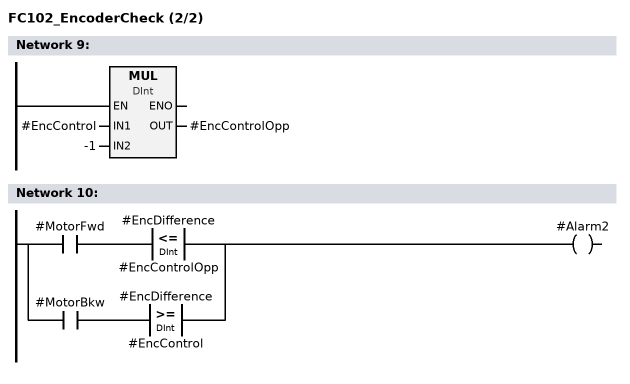
   RUNG wire#powerrail
      { S7_Templates := "SrcType := DInt"; S7_GenerateENO := "TRUE" } Mul(in1 := #EncControl, in2 := -1, out => #EncControlOpp)
   END_RUNG
   // the same network as SCL:
   #EncControlOpp := #EncControl * (-1);
END_REGION

REGION Network 10
   RUNG wire#powerrail
      Contact( #MotorFwd )
      { S7_Templates := "SrcType := DInt" } LE_Contact(in1 := #EncDifference, in2 := #EncControlOpp)
      wire#w1
      Coil( #Alarm2 )
   END_RUNG
   RUNG wire#powerrail
      Contact( #MotorBkw )
      { S7_Templates := "SrcType := DInt" } GE_Contact(in1 := #EncDifference, in2 := #EncControl)
   END_RUNG wire#w1
   // the same network as SCL:
   #Alarm2 := (#MotorFwd AND (#EncDifference <= #EncControlOpp)) OR (#MotorBkw AND (#EncDifference >= #EncControl));
END_REGION
END_FUNCTION

FUNCTION "FC06_TechnoplatCycle" : Void   // FC6, LAD
TITLE = Machine cycle
{ S7_Optimized_Access := 'FALSE' }
AUTHOR : Robopac
VERSION : 0.0
// stored: AutoNumber false, IsIECCheckEnabled false, SetENOAutomatically false, UDAEnableTagReadback false
   VAR_TEMP   // added for the SCL form of the ladder/FBD networks
      _w1 : Bool;
   END_VAR
BEGIN

REGION Network 1: Machine cycle: M0.0 Start cycle
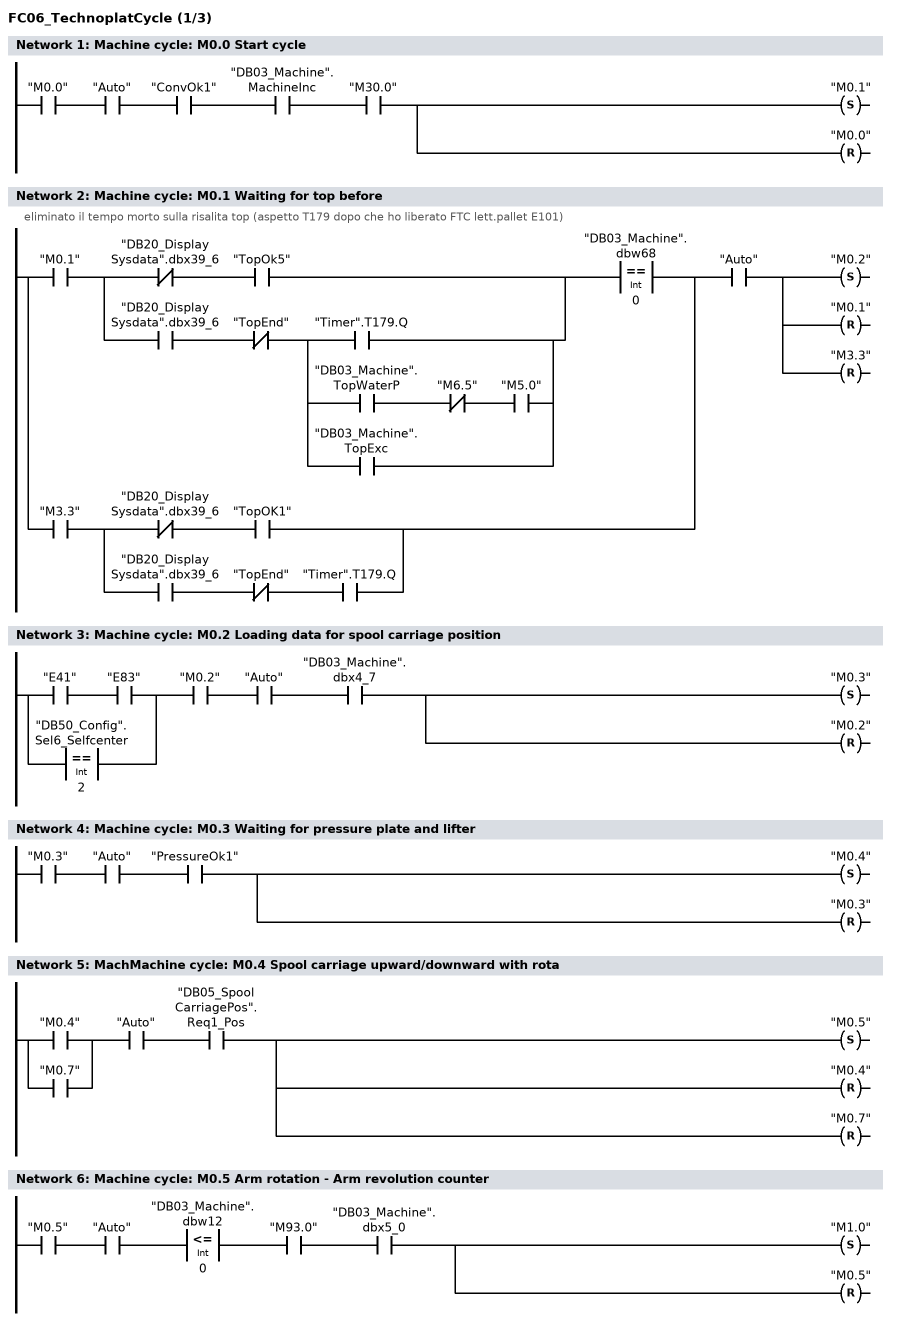
   RUNG wire#powerrail
      Contact( "M0.0" )
      Contact( "Auto" )
      Contact( "ConvOk1" )
      Contact( "DB03_Machine".MachineInc )
      Contact( "M30.0" )
      wire#w1
      S_Coil( "M0.1" )
   END_RUNG
   RUNG wire#w1
      R_Coil( "M0.0" )
   END_RUNG
   // the same network as SCL:
   IF "M0.0" AND "Auto" AND "ConvOk1" AND "DB03_Machine".MachineInc AND "M30.0" THEN
       "M0.1" := TRUE;
       "M0.0" := FALSE;
   END_IF;
END_REGION

REGION Network 2: Machine cycle: M0.1 Waiting for top before
   // eliminato il tempo morto sulla risalita top (aspetto T179 dopo che ho liberato FTC lett.pallet E101)
   RUNG wire#powerrail
      Contact( "M0.1" )
      wire#w1
      I_Contact( "DB20_DisplaySysdata".dbx39_6 )
      Contact( "TopOk5" )
      wire#w2
      { S7_Templates := "SrcType := Int" } EQ_Contact(in1 := "DB03_Machine".dbw68, in2 := 0)
      wire#w4
      Contact( "Auto" )
      wire#w6
      S_Coil( "M0.2" )
   END_RUNG
   RUNG wire#w1
      Contact( "DB20_DisplaySysdata".dbx39_6 )
      I_Contact( "TopEnd" )
      wire#w3
      Contact( "Timer".T179.Q )
   END_RUNG wire#w2
   RUNG wire#w3
      Contact( "DB03_Machine".TopWaterP )
      I_Contact( "M6.5" )
      Contact( "M5.0" )
   END_RUNG wire#w2
   RUNG wire#w3
      Contact( "DB03_Machine".TopExc )
   END_RUNG wire#w2
   RUNG wire#powerrail
      Contact( "M3.3" )
      wire#w5
      I_Contact( "DB20_DisplaySysdata".dbx39_6 )
      Contact( "TopOK1" )
   END_RUNG wire#w4
   RUNG wire#w5
      Contact( "DB20_DisplaySysdata".dbx39_6 )
      I_Contact( "TopEnd" )
      Contact( "Timer".T179.Q )
   END_RUNG wire#w4
   RUNG wire#w6
      R_Coil( "M0.1" )
   END_RUNG
   RUNG wire#w6
      R_Coil( "M3.3" )
   END_RUNG
   // the same network as SCL:
   IF (("M0.1" AND ((NOT "DB20_DisplaySysdata".dbx39_6 AND "TopOk5") OR ("DB20_DisplaySysdata".dbx39_6 AND NOT "TopEnd" AND ("Timer".T179.Q OR ("DB03_Machine".TopWaterP AND NOT "M6.5" AND "M5.0") OR "DB03_Machine".TopExc))) AND ("DB03_Machine".dbw68 = 0)) OR ("M3.3" AND ((NOT "DB20_DisplaySysdata".dbx39_6 AND "TopOK1") OR ("DB20_DisplaySysdata".dbx39_6 AND NOT "TopEnd" AND "Timer".T179.Q)))) AND "Auto" THEN
       "M0.2" := TRUE;
   END_IF;
   #_w1 := (("M0.1" AND ((NOT "DB20_DisplaySysdata".dbx39_6 AND "TopOk5") OR ("DB20_DisplaySysdata".dbx39_6 AND NOT "TopEnd" AND ("Timer".T179.Q OR ("DB03_Machine".TopWaterP AND NOT "M6.5" AND "M5.0") OR "DB03_Machine".TopExc))) AND ("DB03_Machine".dbw68 = 0)) OR ("M3.3" AND ((NOT "DB20_DisplaySysdata".dbx39_6 AND "TopOK1") OR ("DB20_DisplaySysdata".dbx39_6 AND NOT "TopEnd" AND "Timer".T179.Q)))) AND "Auto";
   IF #_w1 THEN
       "M0.1" := FALSE;
       "M3.3" := FALSE;
   END_IF;
END_REGION

REGION Network 3: Machine cycle: M0.2 Loading data for spool carriage position
   RUNG wire#powerrail
      Contact( "E41" )
      Contact( "E83" )
      wire#w1
      Contact( "M0.2" )
      Contact( "Auto" )
      Contact( "DB03_Machine".dbx4_7 )
      wire#w2
      S_Coil( "M0.3" )
   END_RUNG
   RUNG wire#powerrail
      { S7_Templates := "SrcType := Int" } EQ_Contact(in1 := "DB50_Config".Sel6_Selfcenter, in2 := 2)
   END_RUNG wire#w1
   RUNG wire#w2
      R_Coil( "M0.2" )
   END_RUNG
   // the same network as SCL:
   IF (("E41" AND "E83") OR ("DB50_Config".Sel6_Selfcenter = 2)) AND "M0.2" AND "Auto" AND "DB03_Machine".dbx4_7 THEN
       "M0.3" := TRUE;
       "M0.2" := FALSE;
   END_IF;
END_REGION

REGION Network 4: Machine cycle: M0.3 Waiting for pressure plate and lifter
   RUNG wire#powerrail
      Contact( "M0.3" )
      Contact( "Auto" )
      Contact( "PressureOk1" )
      wire#w1
      S_Coil( "M0.4" )
   END_RUNG
   RUNG wire#w1
      R_Coil( "M0.3" )
   END_RUNG
   // the same network as SCL:
   IF "M0.3" AND "Auto" AND "PressureOk1" THEN
       "M0.4" := TRUE;
       "M0.3" := FALSE;
   END_IF;
END_REGION

REGION Network 5: MachMachine cycle: M0.4 Spool carriage upward/downward with rota
   RUNG wire#powerrail
      Contact( "M0.4" )
      wire#w1
      Contact( "Auto" )
      Contact( "DB05_SpoolCarriagePos".Req1_Pos )
      wire#w2
      S_Coil( "M0.5" )
   END_RUNG
   RUNG wire#powerrail
      Contact( "M0.7" )
   END_RUNG wire#w1
   RUNG wire#w2
      R_Coil( "M0.4" )
   END_RUNG
   RUNG wire#w2
      R_Coil( "M0.7" )
   END_RUNG
   // the same network as SCL:
   IF ("M0.4" OR "M0.7") AND "Auto" AND "DB05_SpoolCarriagePos".Req1_Pos THEN "M0.5" := TRUE; END_IF;
   #_w1 := ("M0.4" OR "M0.7") AND "Auto" AND "DB05_SpoolCarriagePos".Req1_Pos;
   IF #_w1 THEN
       "M0.4" := FALSE;
       "M0.7" := FALSE;
   END_IF;
END_REGION

REGION Network 6: Machine cycle: M0.5 Arm rotation - Arm revolution counter
   RUNG wire#powerrail
      Contact( "M0.5" )
      Contact( "Auto" )
      { S7_Templates := "SrcType := Int" } LE_Contact(in1 := "DB03_Machine".dbw12, in2 := 0)
      Contact( "M93.0" )
      Contact( "DB03_Machine".dbx5_0 )
      wire#w1
      S_Coil( "M1.0" )
   END_RUNG
   RUNG wire#w1
      R_Coil( "M0.5" )
   END_RUNG
   // the same network as SCL:
   IF "M0.5" AND "Auto" AND ("DB03_Machine".dbw12 <= 0) AND "M93.0" AND "DB03_Machine".dbx5_0 THEN
       "M1.0" := TRUE;
       "M0.5" := FALSE;
   END_IF;
END_REGION

REGION Network 7: Machine cycle: M1.0 Revolution over welder contrast
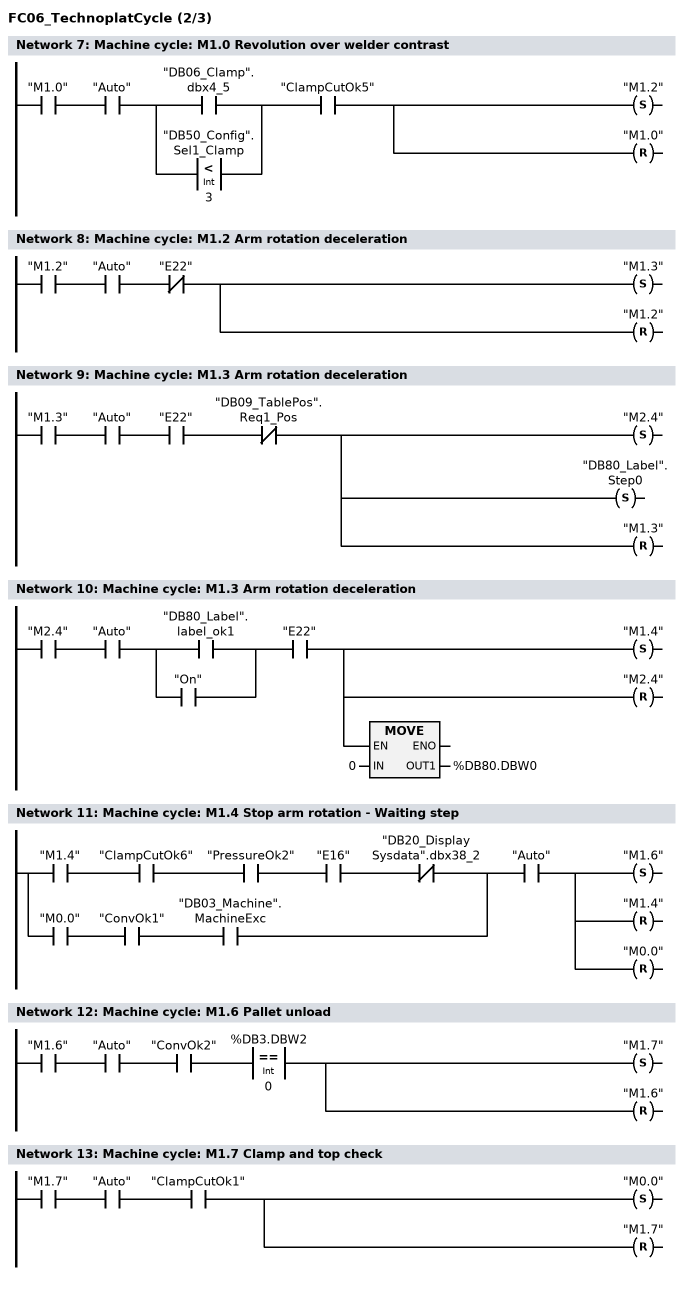
   RUNG wire#powerrail
      Contact( "M1.0" )
      Contact( "Auto" )
      wire#w1
      Contact( "DB06_Clamp".dbx4_5 )
      wire#w2
      Contact( "ClampCutOk5" )
      wire#w3
      S_Coil( "M1.2" )
   END_RUNG
   RUNG wire#w1
      { S7_Templates := "SrcType := Int" } LT_Contact(in1 := "DB50_Config".Sel1_Clamp, in2 := 3)
   END_RUNG wire#w2
   RUNG wire#w3
      R_Coil( "M1.0" )
   END_RUNG
   // the same network as SCL:
   IF "M1.0" AND "Auto" AND ("DB06_Clamp".dbx4_5 OR ("DB50_Config".Sel1_Clamp < 3)) AND "ClampCutOk5" THEN
       "M1.2" := TRUE;
       "M1.0" := FALSE;
   END_IF;
END_REGION

REGION Network 8: Machine cycle: M1.2 Arm rotation deceleration
   RUNG wire#powerrail
      Contact( "M1.2" )
      Contact( "Auto" )
      I_Contact( "E22" )
      wire#w1
      S_Coil( "M1.3" )
   END_RUNG
   RUNG wire#w1
      R_Coil( "M1.2" )
   END_RUNG
   // the same network as SCL:
   IF "M1.2" AND "Auto" AND NOT "E22" THEN
       "M1.3" := TRUE;
       "M1.2" := FALSE;
   END_IF;
END_REGION

REGION Network 9: Machine cycle: M1.3 Arm rotation deceleration
   RUNG wire#powerrail
      Contact( "M1.3" )
      Contact( "Auto" )
      Contact( "E22" )
      I_Contact( "DB09_TablePos".Req1_Pos )
      wire#w1
      S_Coil( "M2.4" )
   END_RUNG
   RUNG wire#w1
      S_Coil( "DB80_Label".Step0 )
   END_RUNG
   RUNG wire#w1
      R_Coil( "M1.3" )
   END_RUNG
   // the same network as SCL:
   IF "M1.3" AND "Auto" AND "E22" AND NOT "DB09_TablePos".Req1_Pos THEN
       "M2.4" := TRUE;
       "DB80_Label".Step0 := TRUE;
       "M1.3" := FALSE;
   END_IF;
END_REGION

REGION Network 10: Machine cycle: M1.3 Arm rotation deceleration
   RUNG wire#powerrail
      Contact( "M2.4" )
      Contact( "Auto" )
      wire#w1
      Contact( "DB80_Label".label_ok1 )
      wire#w2
      Contact( "E22" )
      wire#w3
      S_Coil( "M1.4" )
   END_RUNG
   RUNG wire#w1
      Contact( "On" )
   END_RUNG wire#w2
   RUNG wire#w3
      R_Coil( "M2.4" )
   END_RUNG
   RUNG wire#w3
      { S7_GenerateENO := "TRUE" } Move(in := 0, out1 => %DB80.DBW0)
   END_RUNG
   // the same network as SCL:
   IF "M2.4" AND "Auto" AND ("DB80_Label".label_ok1 OR "On") AND "E22" THEN "M1.4" := TRUE; END_IF;
   #_w1 := "M2.4" AND "Auto" AND ("DB80_Label".label_ok1 OR "On") AND "E22";
   IF #_w1 THEN
       "M2.4" := FALSE;
       %DB80.DBW0 := 0;
   END_IF;
END_REGION

REGION Network 11: Machine cycle: M1.4 Stop arm rotation - Waiting step
   RUNG wire#powerrail
      Contact( "M1.4" )
      Contact( "ClampCutOk6" )
      Contact( "PressureOk2" )
      Contact( "E16" )
      I_Contact( "DB20_DisplaySysdata".dbx38_2 )
      wire#w1
      Contact( "Auto" )
      wire#w2
      S_Coil( "M1.6" )
   END_RUNG
   RUNG wire#powerrail
      Contact( "M0.0" )
      Contact( "ConvOk1" )
      Contact( "DB03_Machine".MachineExc )
   END_RUNG wire#w1
   RUNG wire#w2
      R_Coil( "M1.4" )
   END_RUNG
   RUNG wire#w2
      R_Coil( "M0.0" )
   END_RUNG
   // the same network as SCL:
   IF (("M1.4" AND "ClampCutOk6" AND "PressureOk2" AND "E16" AND NOT "DB20_DisplaySysdata".dbx38_2) OR ("M0.0" AND "ConvOk1" AND "DB03_Machine".MachineExc)) AND "Auto" THEN
       "M1.6" := TRUE;
   END_IF;
   #_w1 := (("M1.4" AND "ClampCutOk6" AND "PressureOk2" AND "E16" AND NOT "DB20_DisplaySysdata".dbx38_2) OR ("M0.0" AND "ConvOk1" AND "DB03_Machine".MachineExc)) AND "Auto";
   IF #_w1 THEN
       "M1.4" := FALSE;
       "M0.0" := FALSE;
   END_IF;
END_REGION

REGION Network 12: Machine cycle: M1.6 Pallet unload
   RUNG wire#powerrail
      Contact( "M1.6" )
      Contact( "Auto" )
      Contact( "ConvOk2" )
      { S7_Templates := "SrcType := Int" } EQ_Contact(in1 := %DB3.DBW2, in2 := 0)
      wire#w1
      S_Coil( "M1.7" )
   END_RUNG
   RUNG wire#w1
      R_Coil( "M1.6" )
   END_RUNG
   // the same network as SCL:
   IF "M1.6" AND "Auto" AND "ConvOk2" AND (%DB3.DBW2 = 0) THEN
       "M1.7" := TRUE;
       "M1.6" := FALSE;
   END_IF;
END_REGION

REGION Network 13: Machine cycle: M1.7 Clamp and top check
   RUNG wire#powerrail
      Contact( "M1.7" )
      Contact( "Auto" )
      Contact( "ClampCutOk1" )
      wire#w1
      S_Coil( "M0.0" )
   END_RUNG
   RUNG wire#w1
      R_Coil( "M1.7" )
   END_RUNG
   // the same network as SCL:
   IF "M1.7" AND "Auto" AND "ClampCutOk1" THEN
       "M0.0" := TRUE;
       "M1.7" := FALSE;
   END_IF;
END_REGION

REGION Network 14: Machine cycle: M0.5 Arm rotation - Arm revolution counter
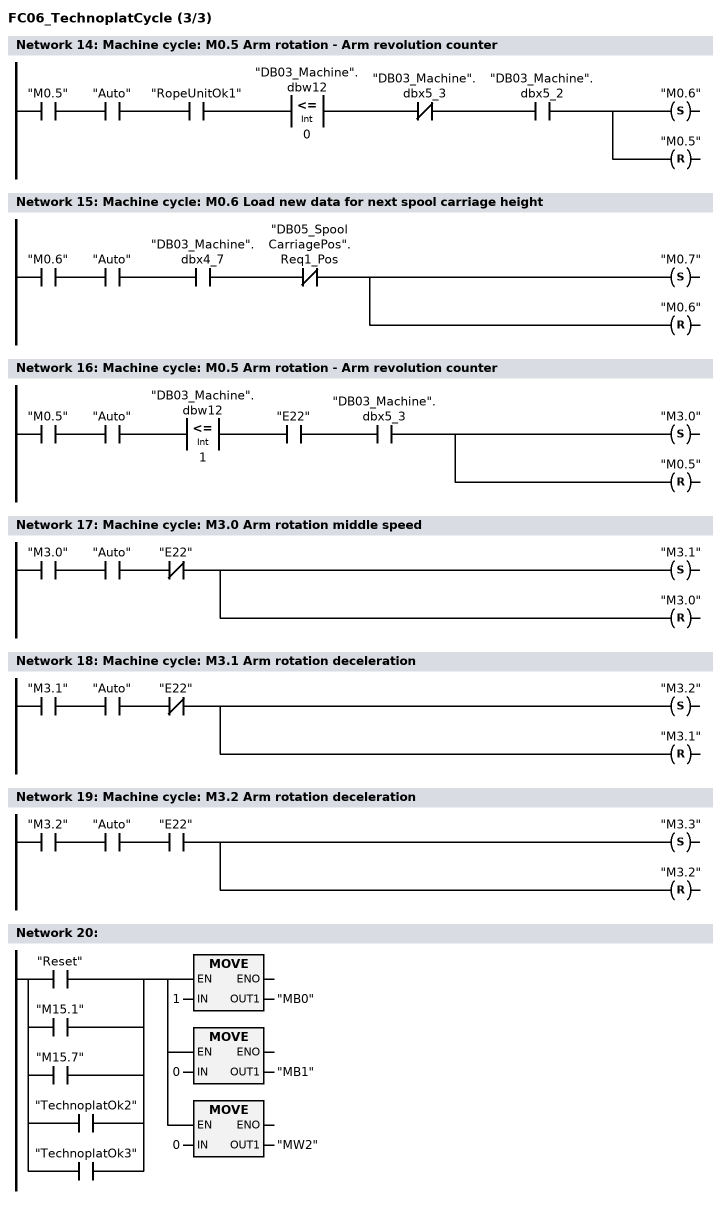
   RUNG wire#powerrail
      Contact( "M0.5" )
      Contact( "Auto" )
      Contact( "RopeUnitOk1" )
      { S7_Templates := "SrcType := Int" } LE_Contact(in1 := "DB03_Machine".dbw12, in2 := 0)
      I_Contact( "DB03_Machine".dbx5_3 )
      Contact( "DB03_Machine".dbx5_2 )
      wire#w1
      S_Coil( "M0.6" )
   END_RUNG
   RUNG wire#w1
      R_Coil( "M0.5" )
   END_RUNG
   // the same network as SCL:
   IF "M0.5" AND "Auto" AND "RopeUnitOk1" AND ("DB03_Machine".dbw12 <= 0) AND NOT "DB03_Machine".dbx5_3 AND "DB03_Machine".dbx5_2 THEN
       "M0.6" := TRUE;
       "M0.5" := FALSE;
   END_IF;
END_REGION

REGION Network 15: Machine cycle: M0.6 Load new data for next spool carriage height
   RUNG wire#powerrail
      Contact( "M0.6" )
      Contact( "Auto" )
      Contact( "DB03_Machine".dbx4_7 )
      I_Contact( "DB05_SpoolCarriagePos".Req1_Pos )
      wire#w1
      S_Coil( "M0.7" )
   END_RUNG
   RUNG wire#w1
      R_Coil( "M0.6" )
   END_RUNG
   // the same network as SCL:
   IF "M0.6" AND "Auto" AND "DB03_Machine".dbx4_7 AND NOT "DB05_SpoolCarriagePos".Req1_Pos THEN
       "M0.7" := TRUE;
       "M0.6" := FALSE;
   END_IF;
END_REGION

REGION Network 16: Machine cycle: M0.5 Arm rotation - Arm revolution counter
   RUNG wire#powerrail
      Contact( "M0.5" )
      Contact( "Auto" )
      { S7_Templates := "SrcType := Int" } LE_Contact(in1 := "DB03_Machine".dbw12, in2 := 1)
      Contact( "E22" )
      Contact( "DB03_Machine".dbx5_3 )
      wire#w1
      S_Coil( "M3.0" )
   END_RUNG
   RUNG wire#w1
      R_Coil( "M0.5" )
   END_RUNG
   // the same network as SCL:
   IF "M0.5" AND "Auto" AND ("DB03_Machine".dbw12 <= 1) AND "E22" AND "DB03_Machine".dbx5_3 THEN
       "M3.0" := TRUE;
       "M0.5" := FALSE;
   END_IF;
END_REGION

REGION Network 17: Machine cycle: M3.0 Arm rotation middle speed
   RUNG wire#powerrail
      Contact( "M3.0" )
      Contact( "Auto" )
      I_Contact( "E22" )
      wire#w1
      S_Coil( "M3.1" )
   END_RUNG
   RUNG wire#w1
      R_Coil( "M3.0" )
   END_RUNG
   // the same network as SCL:
   IF "M3.0" AND "Auto" AND NOT "E22" THEN
       "M3.1" := TRUE;
       "M3.0" := FALSE;
   END_IF;
END_REGION

REGION Network 18: Machine cycle: M3.1 Arm rotation deceleration
   RUNG wire#powerrail
      Contact( "M3.1" )
      Contact( "Auto" )
      I_Contact( "E22" )
      wire#w1
      S_Coil( "M3.2" )
   END_RUNG
   RUNG wire#w1
      R_Coil( "M3.1" )
   END_RUNG
   // the same network as SCL:
   IF "M3.1" AND "Auto" AND NOT "E22" THEN
       "M3.2" := TRUE;
       "M3.1" := FALSE;
   END_IF;
END_REGION

REGION Network 19: Machine cycle: M3.2 Arm rotation deceleration
   RUNG wire#powerrail
      Contact( "M3.2" )
      Contact( "Auto" )
      Contact( "E22" )
      wire#w1
      S_Coil( "M3.3" )
   END_RUNG
   RUNG wire#w1
      R_Coil( "M3.2" )
   END_RUNG
   // the same network as SCL:
   IF "M3.2" AND "Auto" AND "E22" THEN
       "M3.3" := TRUE;
       "M3.2" := FALSE;
   END_IF;
END_REGION

REGION Network 20
   RUNG wire#powerrail
      Contact( "Reset" )
      wire#w1
      { S7_GenerateENO := "TRUE" } Move(in := 1, out1 => "MB0")
   END_RUNG
   RUNG wire#powerrail
      Contact( "M15.1" )
   END_RUNG wire#w1
   RUNG wire#powerrail
      Contact( "M15.7" )
   END_RUNG wire#w1
   RUNG wire#powerrail
      Contact( "TechnoplatOk2" )
   END_RUNG wire#w1
   RUNG wire#powerrail
      Contact( "TechnoplatOk3" )
   END_RUNG wire#w1
   RUNG wire#w1
      { S7_GenerateENO := "TRUE" } Move(in := 0, out1 => "MB1")
   END_RUNG
   RUNG wire#w1
      { S7_GenerateENO := "TRUE" } Move(in := 0, out1 => "MW2")
   END_RUNG
   // the same network as SCL:
   IF "Reset" OR "M15.1" OR "M15.7" OR "TechnoplatOk2" OR "TechnoplatOk3" THEN
       "MB0" := 1;
       "MB1" := 0;
       "MW2" := 0;
   END_IF;
END_REGION
END_FUNCTION

FUNCTION "FC80_Label" : Void   // FC80, LAD
TITLE = Label device
{ S7_Optimized_Access := 'FALSE' }
VERSION : 0.1
// stored: AutoNumber false, IsIECCheckEnabled false, SetENOAutomatically false, UDAEnableTagReadback false
BEGIN

REGION Network 1: Label arm in home position for pallet transit
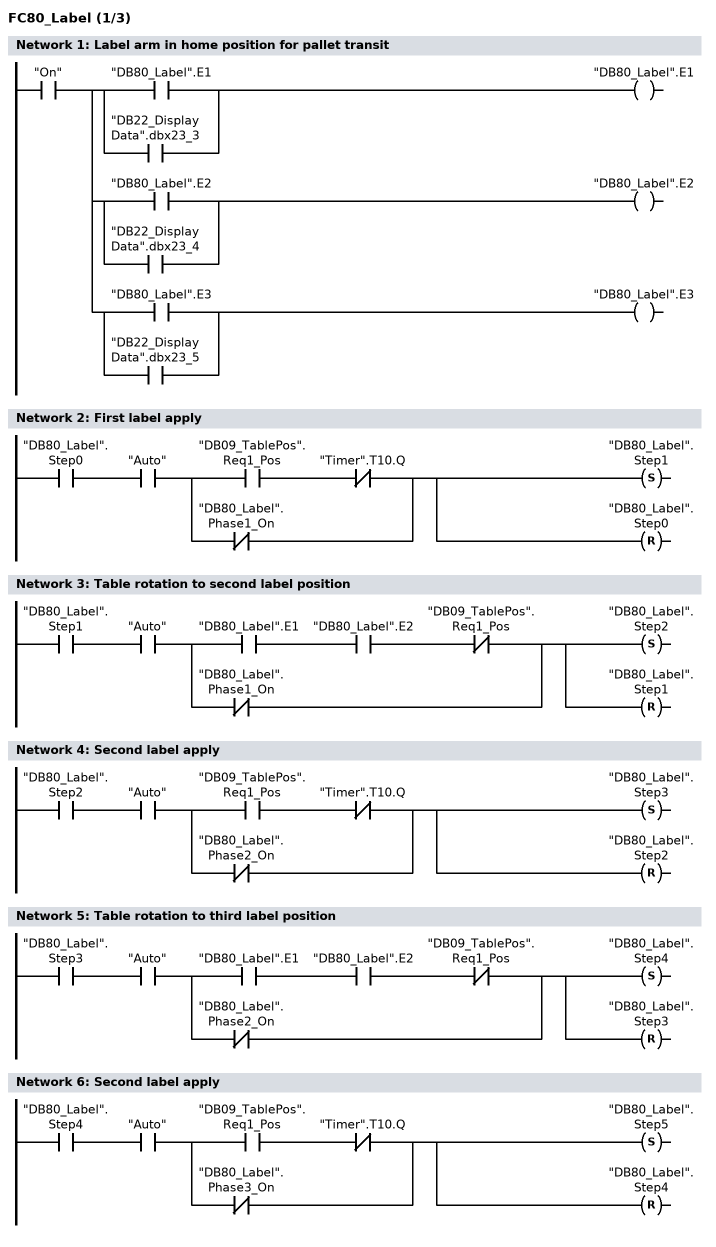
   RUNG wire#powerrail
      Contact( "On" )
      wire#w1
      Contact( "DB80_Label".E1 )
      wire#w2
      Coil( "DB80_Label".E1 )
   END_RUNG
   RUNG wire#w1
      Contact( "DB22_DisplayData".dbx23_3 )
   END_RUNG wire#w2
   RUNG wire#w1
      Contact( "DB80_Label".E2 )
      wire#w3
      Coil( "DB80_Label".E2 )
   END_RUNG
   RUNG wire#w1
      Contact( "DB22_DisplayData".dbx23_4 )
   END_RUNG wire#w3
   RUNG wire#w1
      Contact( "DB80_Label".E3 )
      wire#w4
      Coil( "DB80_Label".E3 )
   END_RUNG
   RUNG wire#w1
      Contact( "DB22_DisplayData".dbx23_5 )
   END_RUNG wire#w4
   // the same network as SCL:
   "DB80_Label".E1 := "On" AND ("DB80_Label".E1 OR "DB22_DisplayData".dbx23_3);
   "DB80_Label".E2 := "On" AND ("DB80_Label".E2 OR "DB22_DisplayData".dbx23_4);
   "DB80_Label".E3 := "On" AND ("DB80_Label".E3 OR "DB22_DisplayData".dbx23_5);
END_REGION

REGION Network 2: First label apply
   RUNG wire#powerrail
      Contact( "DB80_Label".Step0 )
      Contact( "Auto" )
      wire#w1
      Contact( "DB09_TablePos".Req1_Pos )
      I_Contact( "Timer".T10.Q )
      wire#w2
      S_Coil( "DB80_Label".Step1 )
   END_RUNG
   RUNG wire#w1
      I_Contact( "DB80_Label".Phase1_On )
   END_RUNG wire#w2
   RUNG wire#w2
      R_Coil( "DB80_Label".Step0 )
   END_RUNG
   // the same network as SCL:
   IF "DB80_Label".Step0 AND "Auto" AND (("DB09_TablePos".Req1_Pos AND NOT "Timer".T10.Q) OR NOT "DB80_Label".Phase1_On) THEN
       "DB80_Label".Step1 := TRUE;
       "DB80_Label".Step0 := FALSE;
   END_IF;
END_REGION

REGION Network 3: Table rotation to second label position
   RUNG wire#powerrail
      Contact( "DB80_Label".Step1 )
      Contact( "Auto" )
      wire#w1
      Contact( "DB80_Label".E1 )
      Contact( "DB80_Label".E2 )
      I_Contact( "DB09_TablePos".Req1_Pos )
      wire#w2
      S_Coil( "DB80_Label".Step2 )
   END_RUNG
   RUNG wire#w1
      I_Contact( "DB80_Label".Phase1_On )
   END_RUNG wire#w2
   RUNG wire#w2
      R_Coil( "DB80_Label".Step1 )
   END_RUNG
   // the same network as SCL:
   IF "DB80_Label".Step1 AND "Auto" AND (("DB80_Label".E1 AND "DB80_Label".E2 AND NOT "DB09_TablePos".Req1_Pos) OR NOT "DB80_Label".Phase1_On) THEN
       "DB80_Label".Step2 := TRUE;
       "DB80_Label".Step1 := FALSE;
   END_IF;
END_REGION

REGION Network 4: Second label apply
   RUNG wire#powerrail
      Contact( "DB80_Label".Step2 )
      Contact( "Auto" )
      wire#w1
      Contact( "DB09_TablePos".Req1_Pos )
      I_Contact( "Timer".T10.Q )
      wire#w2
      S_Coil( "DB80_Label".Step3 )
   END_RUNG
   RUNG wire#w1
      I_Contact( "DB80_Label".Phase2_On )
   END_RUNG wire#w2
   RUNG wire#w2
      R_Coil( "DB80_Label".Step2 )
   END_RUNG
   // the same network as SCL:
   IF "DB80_Label".Step2 AND "Auto" AND (("DB09_TablePos".Req1_Pos AND NOT "Timer".T10.Q) OR NOT "DB80_Label".Phase2_On) THEN
       "DB80_Label".Step3 := TRUE;
       "DB80_Label".Step2 := FALSE;
   END_IF;
END_REGION

REGION Network 5: Table rotation to third label position
   RUNG wire#powerrail
      Contact( "DB80_Label".Step3 )
      Contact( "Auto" )
      wire#w1
      Contact( "DB80_Label".E1 )
      Contact( "DB80_Label".E2 )
      I_Contact( "DB09_TablePos".Req1_Pos )
      wire#w2
      S_Coil( "DB80_Label".Step4 )
   END_RUNG
   RUNG wire#w1
      I_Contact( "DB80_Label".Phase2_On )
   END_RUNG wire#w2
   RUNG wire#w2
      R_Coil( "DB80_Label".Step3 )
   END_RUNG
   // the same network as SCL:
   IF "DB80_Label".Step3 AND "Auto" AND (("DB80_Label".E1 AND "DB80_Label".E2 AND NOT "DB09_TablePos".Req1_Pos) OR NOT "DB80_Label".Phase2_On) THEN
       "DB80_Label".Step4 := TRUE;
       "DB80_Label".Step3 := FALSE;
   END_IF;
END_REGION

REGION Network 6: Second label apply
   RUNG wire#powerrail
      Contact( "DB80_Label".Step4 )
      Contact( "Auto" )
      wire#w1
      Contact( "DB09_TablePos".Req1_Pos )
      I_Contact( "Timer".T10.Q )
      wire#w2
      S_Coil( "DB80_Label".Step5 )
   END_RUNG
   RUNG wire#w1
      I_Contact( "DB80_Label".Phase3_On )
   END_RUNG wire#w2
   RUNG wire#w2
      R_Coil( "DB80_Label".Step4 )
   END_RUNG
   // the same network as SCL:
   IF "DB80_Label".Step4 AND "Auto" AND (("DB09_TablePos".Req1_Pos AND NOT "Timer".T10.Q) OR NOT "DB80_Label".Phase3_On) THEN
       "DB80_Label".Step5 := TRUE;
       "DB80_Label".Step4 := FALSE;
   END_IF;
END_REGION

REGION Network 7: Table rotation to fourth label position
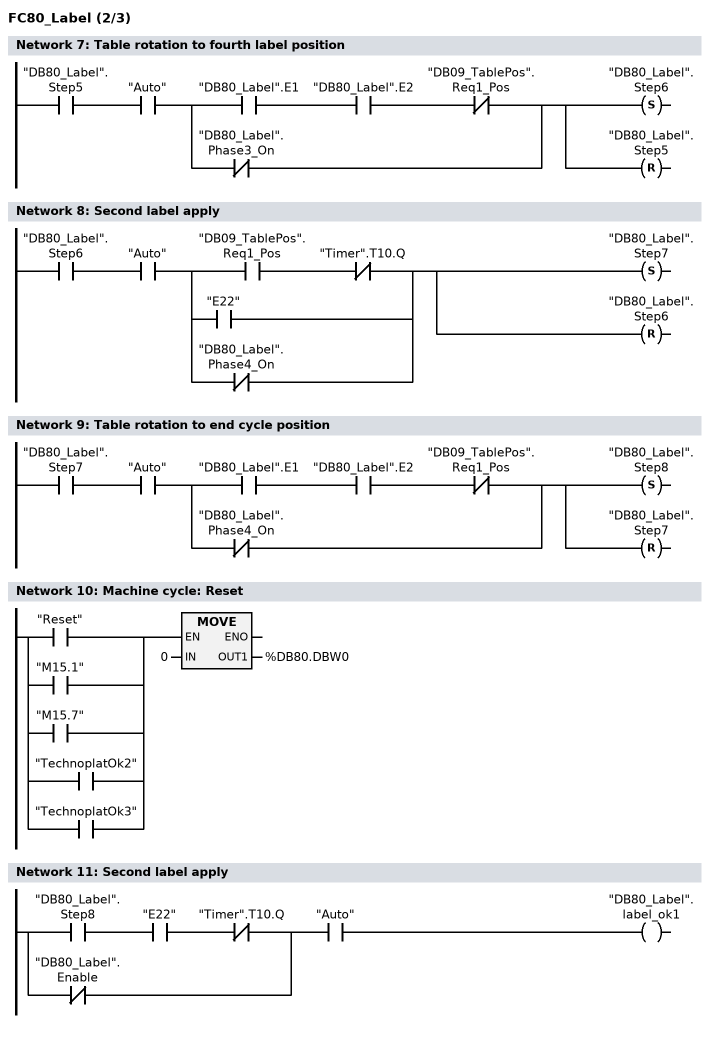
   RUNG wire#powerrail
      Contact( "DB80_Label".Step5 )
      Contact( "Auto" )
      wire#w1
      Contact( "DB80_Label".E1 )
      Contact( "DB80_Label".E2 )
      I_Contact( "DB09_TablePos".Req1_Pos )
      wire#w2
      S_Coil( "DB80_Label".Step6 )
   END_RUNG
   RUNG wire#w1
      I_Contact( "DB80_Label".Phase3_On )
   END_RUNG wire#w2
   RUNG wire#w2
      R_Coil( "DB80_Label".Step5 )
   END_RUNG
   // the same network as SCL:
   IF "DB80_Label".Step5 AND "Auto" AND (("DB80_Label".E1 AND "DB80_Label".E2 AND NOT "DB09_TablePos".Req1_Pos) OR NOT "DB80_Label".Phase3_On) THEN
       "DB80_Label".Step6 := TRUE;
       "DB80_Label".Step5 := FALSE;
   END_IF;
END_REGION

REGION Network 8: Second label apply
   RUNG wire#powerrail
      Contact( "DB80_Label".Step6 )
      Contact( "Auto" )
      wire#w1
      Contact( "DB09_TablePos".Req1_Pos )
      I_Contact( "Timer".T10.Q )
      wire#w2
      S_Coil( "DB80_Label".Step7 )
   END_RUNG
   RUNG wire#w1
      Contact( "E22" )
   END_RUNG wire#w2
   RUNG wire#w1
      I_Contact( "DB80_Label".Phase4_On )
   END_RUNG wire#w2
   RUNG wire#w2
      R_Coil( "DB80_Label".Step6 )
   END_RUNG
   // the same network as SCL:
   IF "DB80_Label".Step6 AND "Auto" AND (("DB09_TablePos".Req1_Pos AND NOT "Timer".T10.Q) OR "E22" OR NOT "DB80_Label".Phase4_On) THEN
       "DB80_Label".Step7 := TRUE;
       "DB80_Label".Step6 := FALSE;
   END_IF;
END_REGION

REGION Network 9: Table rotation to end cycle position
   RUNG wire#powerrail
      Contact( "DB80_Label".Step7 )
      Contact( "Auto" )
      wire#w1
      Contact( "DB80_Label".E1 )
      Contact( "DB80_Label".E2 )
      I_Contact( "DB09_TablePos".Req1_Pos )
      wire#w2
      S_Coil( "DB80_Label".Step8 )
   END_RUNG
   RUNG wire#w1
      I_Contact( "DB80_Label".Phase4_On )
   END_RUNG wire#w2
   RUNG wire#w2
      R_Coil( "DB80_Label".Step7 )
   END_RUNG
   // the same network as SCL:
   IF "DB80_Label".Step7 AND "Auto" AND (("DB80_Label".E1 AND "DB80_Label".E2 AND NOT "DB09_TablePos".Req1_Pos) OR NOT "DB80_Label".Phase4_On) THEN
       "DB80_Label".Step8 := TRUE;
       "DB80_Label".Step7 := FALSE;
   END_IF;
END_REGION

REGION Network 10: Machine cycle: Reset
   RUNG wire#powerrail
      Contact( "Reset" )
      wire#w1
      { S7_GenerateENO := "TRUE" } Move(in := 0, out1 => %DB80.DBW0)
   END_RUNG
   RUNG wire#powerrail
      Contact( "M15.1" )
   END_RUNG wire#w1
   RUNG wire#powerrail
      Contact( "M15.7" )
   END_RUNG wire#w1
   RUNG wire#powerrail
      Contact( "TechnoplatOk2" )
   END_RUNG wire#w1
   RUNG wire#powerrail
      Contact( "TechnoplatOk3" )
   END_RUNG wire#w1
   // the same network as SCL:
   IF "Reset" OR "M15.1" OR "M15.7" OR "TechnoplatOk2" OR "TechnoplatOk3" THEN %DB80.DBW0 := 0; END_IF;
END_REGION

REGION Network 11: Second label apply
   RUNG wire#powerrail
      Contact( "DB80_Label".Step8 )
      Contact( "E22" )
      I_Contact( "Timer".T10.Q )
      wire#w1
      Contact( "Auto" )
      Coil( "DB80_Label".label_ok1 )
   END_RUNG
   RUNG wire#powerrail
      I_Contact( "DB80_Label".Enable )
   END_RUNG wire#w1
   // the same network as SCL:
   "DB80_Label".label_ok1 := (("DB80_Label".Step8 AND "E22" AND NOT "Timer".T10.Q) OR NOT "DB80_Label".Enable) AND "Auto";
END_REGION

REGION Network 12: Label phases
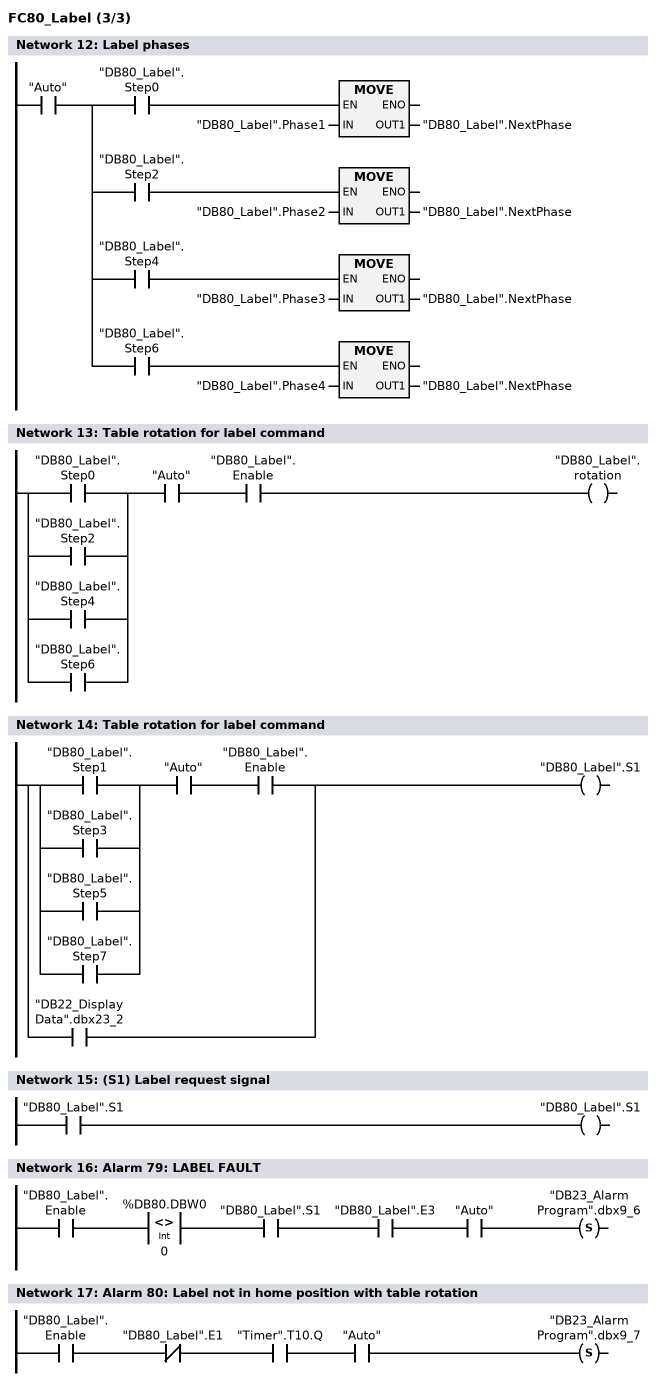
   RUNG wire#powerrail
      Contact( "Auto" )
      wire#w1
      Contact( "DB80_Label".Step0 )
      { S7_GenerateENO := "TRUE" } Move(in := "DB80_Label".Phase1, out1 => "DB80_Label".NextPhase)
   END_RUNG
   RUNG wire#w1
      Contact( "DB80_Label".Step2 )
      { S7_GenerateENO := "TRUE" } Move(in := "DB80_Label".Phase2, out1 => "DB80_Label".NextPhase)
   END_RUNG
   RUNG wire#w1
      Contact( "DB80_Label".Step4 )
      { S7_GenerateENO := "TRUE" } Move(in := "DB80_Label".Phase3, out1 => "DB80_Label".NextPhase)
   END_RUNG
   RUNG wire#w1
      Contact( "DB80_Label".Step6 )
      { S7_GenerateENO := "TRUE" } Move(in := "DB80_Label".Phase4, out1 => "DB80_Label".NextPhase)
   END_RUNG
   // the same network as SCL:
   IF "Auto" AND "DB80_Label".Step0 THEN "DB80_Label".NextPhase := "DB80_Label".Phase1; END_IF;
   IF "Auto" AND "DB80_Label".Step2 THEN "DB80_Label".NextPhase := "DB80_Label".Phase2; END_IF;
   IF "Auto" AND "DB80_Label".Step4 THEN "DB80_Label".NextPhase := "DB80_Label".Phase3; END_IF;
   IF "Auto" AND "DB80_Label".Step6 THEN "DB80_Label".NextPhase := "DB80_Label".Phase4; END_IF;
END_REGION

REGION Network 13: Table rotation for label command
   RUNG wire#powerrail
      Contact( "DB80_Label".Step0 )
      wire#w1
      Contact( "Auto" )
      Contact( "DB80_Label".Enable )
      Coil( "DB80_Label".rotation )
   END_RUNG
   RUNG wire#powerrail
      Contact( "DB80_Label".Step2 )
   END_RUNG wire#w1
   RUNG wire#powerrail
      Contact( "DB80_Label".Step4 )
   END_RUNG wire#w1
   RUNG wire#powerrail
      Contact( "DB80_Label".Step6 )
   END_RUNG wire#w1
   // the same network as SCL:
   "DB80_Label".rotation := ("DB80_Label".Step0 OR "DB80_Label".Step2 OR "DB80_Label".Step4 OR "DB80_Label".Step6) AND "Auto" AND "DB80_Label".Enable;
END_REGION

REGION Network 14: Table rotation for label command
   RUNG wire#powerrail
      Contact( "DB80_Label".Step1 )
      wire#w1
      Contact( "Auto" )
      Contact( "DB80_Label".Enable )
      wire#w2
      Coil( "DB80_Label".S1 )
   END_RUNG
   RUNG wire#powerrail
      Contact( "DB80_Label".Step3 )
   END_RUNG wire#w1
   RUNG wire#powerrail
      Contact( "DB80_Label".Step5 )
   END_RUNG wire#w1
   RUNG wire#powerrail
      Contact( "DB80_Label".Step7 )
   END_RUNG wire#w1
   RUNG wire#powerrail
      Contact( "DB22_DisplayData".dbx23_2 )
   END_RUNG wire#w2
   // the same network as SCL:
   "DB80_Label".S1 := (("DB80_Label".Step1 OR "DB80_Label".Step3 OR "DB80_Label".Step5 OR "DB80_Label".Step7) AND "Auto" AND "DB80_Label".Enable) OR "DB22_DisplayData".dbx23_2;
END_REGION

REGION Network 15: (S1) Label request signal
   RUNG wire#powerrail
      Contact( "DB80_Label".S1 )
      Coil( "DB80_Label".S1 )
   END_RUNG
   // the same network as SCL:
   "DB80_Label".S1 := "DB80_Label".S1;
END_REGION

REGION Network 16: Alarm 79: LABEL FAULT
   RUNG wire#powerrail
      Contact( "DB80_Label".Enable )
      { S7_Templates := "SrcType := Int" } NE_Contact(in1 := %DB80.DBW0, in2 := 0)
      Contact( "DB80_Label".S1 )
      Contact( "DB80_Label".E3 )
      Contact( "Auto" )
      S_Coil( "DB23_AlarmProgram".dbx9_6 )
   END_RUNG
   // the same network as SCL:
   IF "DB80_Label".Enable AND (%DB80.DBW0 <> 0) AND "DB80_Label".S1 AND "DB80_Label".E3 AND "Auto" THEN
       "DB23_AlarmProgram".dbx9_6 := TRUE;
   END_IF;
END_REGION

REGION Network 17: Alarm 80: Label not in home position with table rotation
   RUNG wire#powerrail
      Contact( "DB80_Label".Enable )
      I_Contact( "DB80_Label".E1 )
      Contact( "Timer".T10.Q )
      Contact( "Auto" )
      S_Coil( "DB23_AlarmProgram".dbx9_7 )
   END_RUNG
   // the same network as SCL:
   IF "DB80_Label".Enable AND NOT "DB80_Label".E1 AND "Timer".T10.Q AND "Auto" THEN
       "DB23_AlarmProgram".dbx9_7 := TRUE;
   END_IF;
END_REGION
END_FUNCTION

FUNCTION "FC07_FilmBroken&Test" : Void   // FC7, LAD
TITLE = Film broken or ended management
{ S7_Optimized_Access := 'FALSE' }
AUTHOR : Robopac
VERSION : 0.0
// stored: AutoNumber false, IsIECCheckEnabled false, SetENOAutomatically false, UDAEnableTagReadback false
   VAR_TEMP   // added for the SCL form of the ladder/FBD networks
      _w1 : Bool;
   END_VAR
BEGIN

REGION Network 1: Delay for test cycle
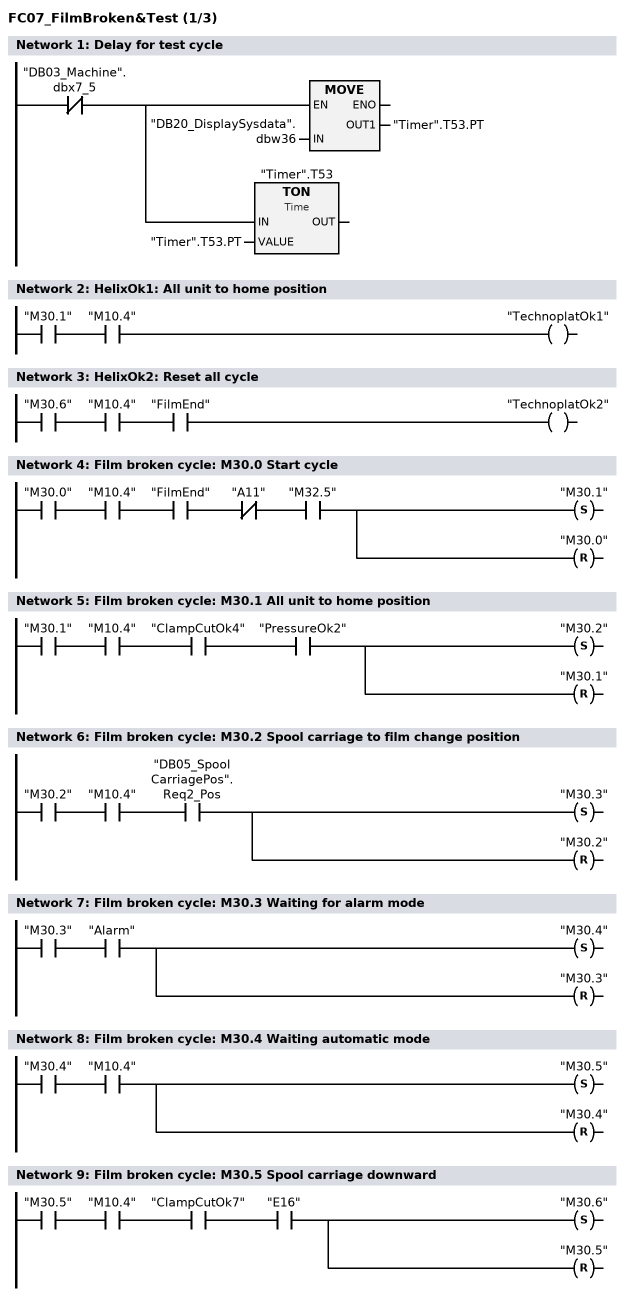
   #_w1 := NOT "DB03_Machine".dbx7_5;
   IF #_w1 THEN "Timer".T53.PT := "DB20_DisplaySysdata".dbw36; END_IF;
   "Timer".T53.TON(IN := #_w1, PT := "Timer".T53.PT);   // TON coil
END_REGION

REGION Network 2: HelixOk1: All unit to home position
   RUNG wire#powerrail
      Contact( "M30.1" )
      Contact( "M10.4" )
      Coil( "TechnoplatOk1" )
   END_RUNG
   // the same network as SCL:
   "TechnoplatOk1" := "M30.1" AND "M10.4";
END_REGION

REGION Network 3: HelixOk2: Reset all cycle
   RUNG wire#powerrail
      Contact( "M30.6" )
      Contact( "M10.4" )
      Contact( "FilmEnd" )
      Coil( "TechnoplatOk2" )
   END_RUNG
   // the same network as SCL:
   "TechnoplatOk2" := "M30.6" AND "M10.4" AND "FilmEnd";
END_REGION

REGION Network 4: Film broken cycle: M30.0 Start cycle
   RUNG wire#powerrail
      Contact( "M30.0" )
      Contact( "M10.4" )
      Contact( "FilmEnd" )
      I_Contact( "A11" )
      Contact( "M32.5" )
      wire#w1
      S_Coil( "M30.1" )
   END_RUNG
   RUNG wire#w1
      R_Coil( "M30.0" )
   END_RUNG
   // the same network as SCL:
   IF "M30.0" AND "M10.4" AND "FilmEnd" AND NOT "A11" AND "M32.5" THEN
       "M30.1" := TRUE;
       "M30.0" := FALSE;
   END_IF;
END_REGION

REGION Network 5: Film broken cycle: M30.1 All unit to home position
   RUNG wire#powerrail
      Contact( "M30.1" )
      Contact( "M10.4" )
      Contact( "ClampCutOk4" )
      Contact( "PressureOk2" )
      wire#w1
      S_Coil( "M30.2" )
   END_RUNG
   RUNG wire#w1
      R_Coil( "M30.1" )
   END_RUNG
   // the same network as SCL:
   IF "M30.1" AND "M10.4" AND "ClampCutOk4" AND "PressureOk2" THEN
       "M30.2" := TRUE;
       "M30.1" := FALSE;
   END_IF;
END_REGION

REGION Network 6: Film broken cycle: M30.2 Spool carriage to film change position
   RUNG wire#powerrail
      Contact( "M30.2" )
      Contact( "M10.4" )
      Contact( "DB05_SpoolCarriagePos".Req2_Pos )
      wire#w1
      S_Coil( "M30.3" )
   END_RUNG
   RUNG wire#w1
      R_Coil( "M30.2" )
   END_RUNG
   // the same network as SCL:
   IF "M30.2" AND "M10.4" AND "DB05_SpoolCarriagePos".Req2_Pos THEN
       "M30.3" := TRUE;
       "M30.2" := FALSE;
   END_IF;
END_REGION

REGION Network 7: Film broken cycle: M30.3 Waiting for alarm mode
   RUNG wire#powerrail
      Contact( "M30.3" )
      Contact( "Alarm" )
      wire#w1
      S_Coil( "M30.4" )
   END_RUNG
   RUNG wire#w1
      R_Coil( "M30.3" )
   END_RUNG
   // the same network as SCL:
   IF "M30.3" AND "Alarm" THEN
       "M30.4" := TRUE;
       "M30.3" := FALSE;
   END_IF;
END_REGION

REGION Network 8: Film broken cycle: M30.4 Waiting automatic mode
   RUNG wire#powerrail
      Contact( "M30.4" )
      Contact( "M10.4" )
      wire#w1
      S_Coil( "M30.5" )
   END_RUNG
   RUNG wire#w1
      R_Coil( "M30.4" )
   END_RUNG
   // the same network as SCL:
   IF "M30.4" AND "M10.4" THEN
       "M30.5" := TRUE;
       "M30.4" := FALSE;
   END_IF;
END_REGION

REGION Network 9: Film broken cycle: M30.5 Spool carriage downward
   RUNG wire#powerrail
      Contact( "M30.5" )
      Contact( "M10.4" )
      Contact( "ClampCutOk7" )
      Contact( "E16" )
      wire#w1
      S_Coil( "M30.6" )
   END_RUNG
   RUNG wire#w1
      R_Coil( "M30.5" )
   END_RUNG
   // the same network as SCL:
   IF "M30.5" AND "M10.4" AND "ClampCutOk7" AND "E16" THEN
       "M30.6" := TRUE;
       "M30.5" := FALSE;
   END_IF;
END_REGION

REGION Network 10: Film broken cycle: M30.6 Waiting step
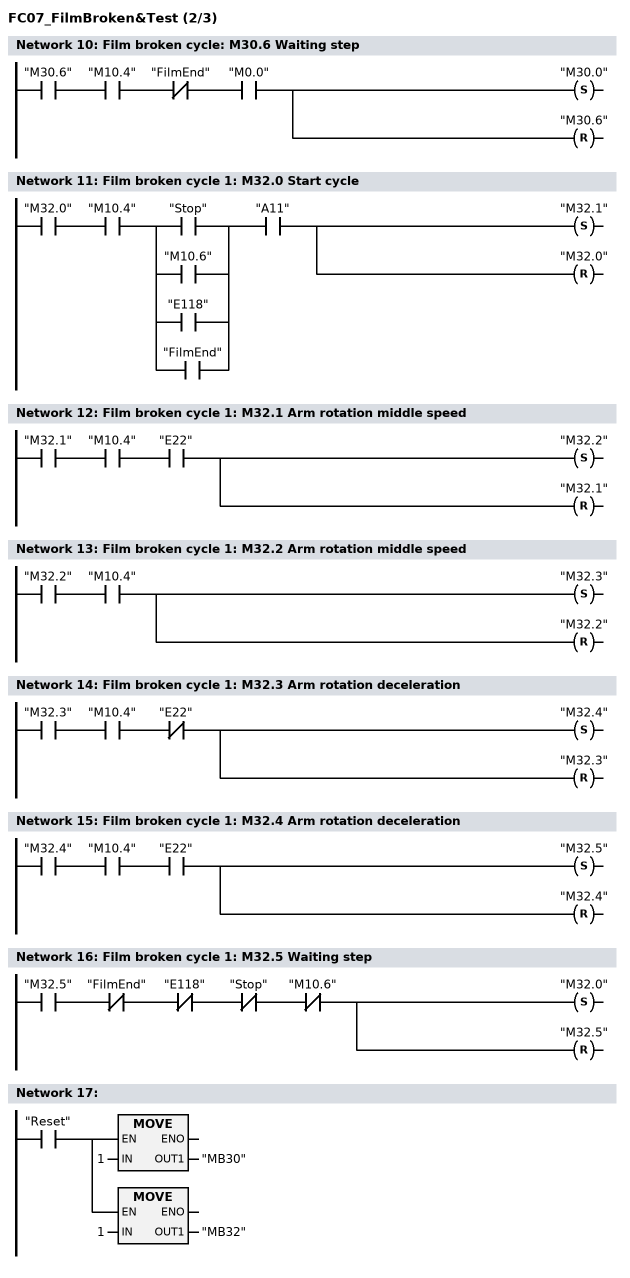
   RUNG wire#powerrail
      Contact( "M30.6" )
      Contact( "M10.4" )
      I_Contact( "FilmEnd" )
      Contact( "M0.0" )
      wire#w1
      S_Coil( "M30.0" )
   END_RUNG
   RUNG wire#w1
      R_Coil( "M30.6" )
   END_RUNG
   // the same network as SCL:
   IF "M30.6" AND "M10.4" AND NOT "FilmEnd" AND "M0.0" THEN
       "M30.0" := TRUE;
       "M30.6" := FALSE;
   END_IF;
END_REGION

REGION Network 11: Film broken cycle 1: M32.0 Start cycle
   RUNG wire#powerrail
      Contact( "M32.0" )
      Contact( "M10.4" )
      wire#w1
      Contact( "Stop" )
      wire#w2
      Contact( "A11" )
      wire#w3
      S_Coil( "M32.1" )
   END_RUNG
   RUNG wire#w1
      Contact( "M10.6" )
   END_RUNG wire#w2
   RUNG wire#w1
      Contact( "E118" )
   END_RUNG wire#w2
   RUNG wire#w1
      Contact( "FilmEnd" )
   END_RUNG wire#w2
   RUNG wire#w3
      R_Coil( "M32.0" )
   END_RUNG
   // the same network as SCL:
   IF "M32.0" AND "M10.4" AND ("Stop" OR "M10.6" OR "E118" OR "FilmEnd") AND "A11" THEN
       "M32.1" := TRUE;
       "M32.0" := FALSE;
   END_IF;
END_REGION

REGION Network 12: Film broken cycle 1: M32.1 Arm rotation middle speed
   RUNG wire#powerrail
      Contact( "M32.1" )
      Contact( "M10.4" )
      Contact( "E22" )
      wire#w1
      S_Coil( "M32.2" )
   END_RUNG
   RUNG wire#w1
      R_Coil( "M32.1" )
   END_RUNG
   // the same network as SCL:
   IF "M32.1" AND "M10.4" AND "E22" THEN
       "M32.2" := TRUE;
       "M32.1" := FALSE;
   END_IF;
END_REGION

REGION Network 13: Film broken cycle 1: M32.2 Arm rotation middle speed
   RUNG wire#powerrail
      Contact( "M32.2" )
      Contact( "M10.4" )
      wire#w1
      S_Coil( "M32.3" )
   END_RUNG
   RUNG wire#w1
      R_Coil( "M32.2" )
   END_RUNG
   // the same network as SCL:
   IF "M32.2" AND "M10.4" THEN
       "M32.3" := TRUE;
       "M32.2" := FALSE;
   END_IF;
END_REGION

REGION Network 14: Film broken cycle 1: M32.3 Arm rotation deceleration
   RUNG wire#powerrail
      Contact( "M32.3" )
      Contact( "M10.4" )
      I_Contact( "E22" )
      wire#w1
      S_Coil( "M32.4" )
   END_RUNG
   RUNG wire#w1
      R_Coil( "M32.3" )
   END_RUNG
   // the same network as SCL:
   IF "M32.3" AND "M10.4" AND NOT "E22" THEN
       "M32.4" := TRUE;
       "M32.3" := FALSE;
   END_IF;
END_REGION

REGION Network 15: Film broken cycle 1: M32.4 Arm rotation deceleration
   RUNG wire#powerrail
      Contact( "M32.4" )
      Contact( "M10.4" )
      Contact( "E22" )
      wire#w1
      S_Coil( "M32.5" )
   END_RUNG
   RUNG wire#w1
      R_Coil( "M32.4" )
   END_RUNG
   // the same network as SCL:
   IF "M32.4" AND "M10.4" AND "E22" THEN
       "M32.5" := TRUE;
       "M32.4" := FALSE;
   END_IF;
END_REGION

REGION Network 16: Film broken cycle 1: M32.5 Waiting step
   RUNG wire#powerrail
      Contact( "M32.5" )
      I_Contact( "FilmEnd" )
      I_Contact( "E118" )
      I_Contact( "Stop" )
      I_Contact( "M10.6" )
      wire#w1
      S_Coil( "M32.0" )
   END_RUNG
   RUNG wire#w1
      R_Coil( "M32.5" )
   END_RUNG
   // the same network as SCL:
   IF "M32.5" AND NOT "FilmEnd" AND NOT "E118" AND NOT "Stop" AND NOT "M10.6" THEN
       "M32.0" := TRUE;
       "M32.5" := FALSE;
   END_IF;
END_REGION

REGION Network 17
   RUNG wire#powerrail
      Contact( "Reset" )
      wire#w1
      { S7_GenerateENO := "TRUE" } Move(in := 1, out1 => "MB30")
   END_RUNG
   RUNG wire#w1
      { S7_GenerateENO := "TRUE" } Move(in := 1, out1 => "MB32")
   END_RUNG
   // the same network as SCL:
   IF "Reset" THEN
       "MB30" := 1;
       "MB32" := 1;
   END_IF;
END_REGION

REGION Network 18: Machine cycle: M1.5 Waiting step
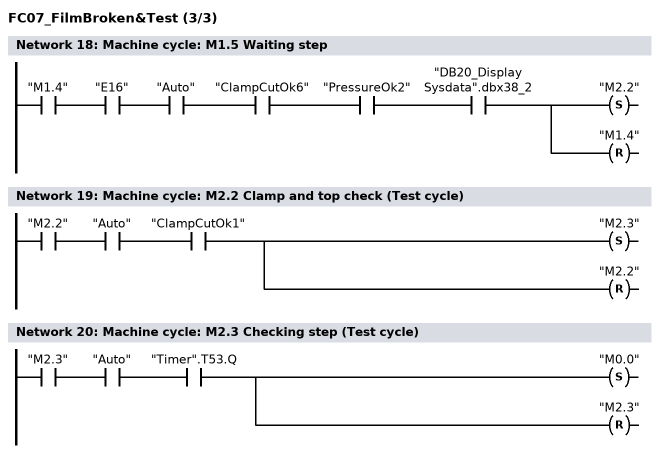
   RUNG wire#powerrail
      Contact( "M1.4" )
      Contact( "E16" )
      Contact( "Auto" )
      Contact( "ClampCutOk6" )
      Contact( "PressureOk2" )
      Contact( "DB20_DisplaySysdata".dbx38_2 )
      wire#w1
      S_Coil( "M2.2" )
   END_RUNG
   RUNG wire#w1
      R_Coil( "M1.4" )
   END_RUNG
   // the same network as SCL:
   IF "M1.4" AND "E16" AND "Auto" AND "ClampCutOk6" AND "PressureOk2" AND "DB20_DisplaySysdata".dbx38_2 THEN
       "M2.2" := TRUE;
       "M1.4" := FALSE;
   END_IF;
END_REGION

REGION Network 19: Machine cycle: M2.2 Clamp and top check (Test cycle)
   RUNG wire#powerrail
      Contact( "M2.2" )
      Contact( "Auto" )
      Contact( "ClampCutOk1" )
      wire#w1
      S_Coil( "M2.3" )
   END_RUNG
   RUNG wire#w1
      R_Coil( "M2.2" )
   END_RUNG
   // the same network as SCL:
   IF "M2.2" AND "Auto" AND "ClampCutOk1" THEN
       "M2.3" := TRUE;
       "M2.2" := FALSE;
   END_IF;
END_REGION

REGION Network 20: Machine cycle: M2.3 Checking step (Test cycle)
   RUNG wire#powerrail
      Contact( "M2.3" )
      Contact( "Auto" )
      Contact( "Timer".T53.Q )
      wire#w1
      S_Coil( "M0.0" )
   END_RUNG
   RUNG wire#w1
      R_Coil( "M2.3" )
   END_RUNG
   // the same network as SCL:
   IF "M2.3" AND "Auto" AND "Timer".T53.Q THEN
       "M0.0" := TRUE;
       "M2.3" := FALSE;
   END_IF;
END_REGION
END_FUNCTION

FUNCTION "Inverter_CW_Assembly" : Void   // FC16, FBD
{ S7_Optimized_Access := 'TRUE' }
VERSION : 0.1
// stored: AutoNumber false, IsIECCheckEnabled false, SetENOAutomatically false, UDAEnableTagReadback false
   VAR_INPUT
      CW_Off1_On : Bool;
      CW_Off2 : Bool;
      CW_Off3 : Bool;
      CW_enable_operation : Bool;
      CW_no_lock_RFG : Bool;
      CW_no_stop_RFG : Bool;
      CW_enable_setpoint : Bool;
      CW_acknowledge : Bool;
      CW_not_used_1 : Bool;
      CW_not_used_2 : Bool;
      CW_PLC_is_Master : Bool;
      CW_direction_reversal : Bool;
      CW_not_used_3 : Bool;
      CW_motortpoti_up : Bool;
      CW_motortpoti_down : Bool;
      CW_not_used_4 : Bool;
   END_VAR
   VAR_IN_OUT
      Control_word : Word;
   END_VAR
BEGIN

REGION Network 1
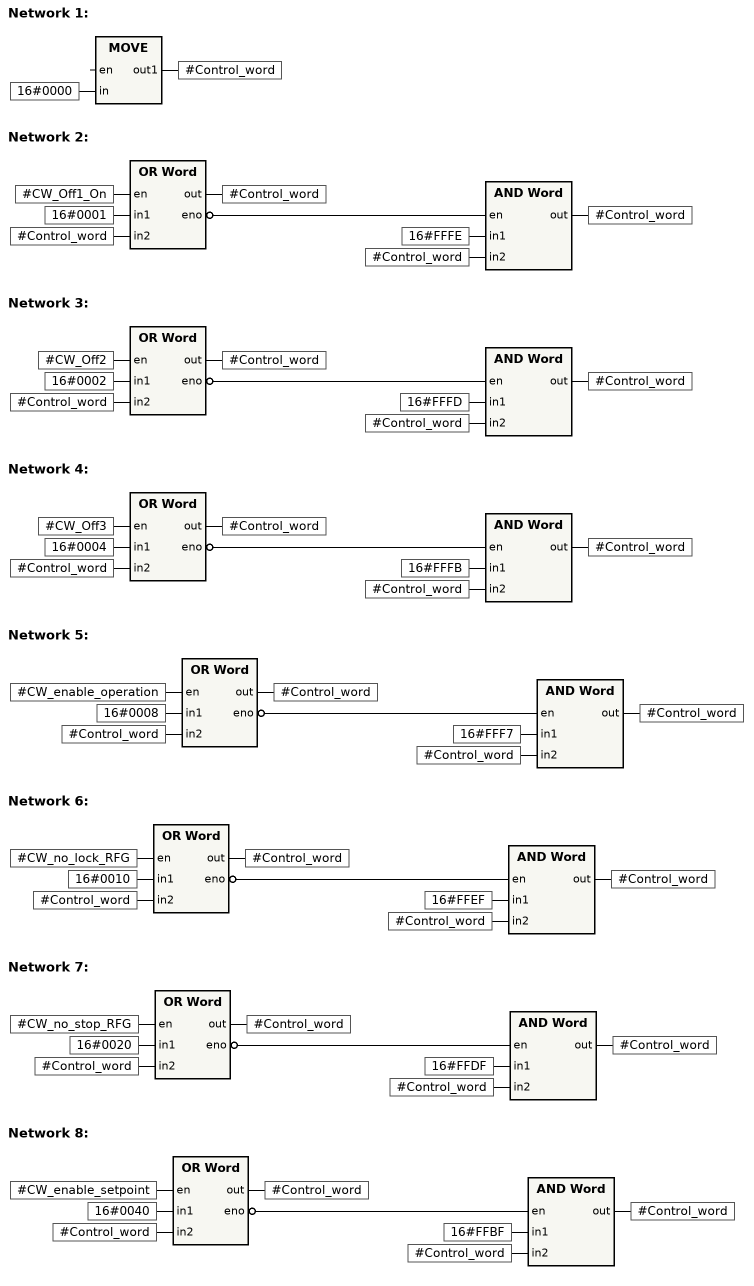
   #Control_word := 16#0000;
END_REGION

REGION Network 2
   IF #CW_Off1_On THEN #Control_word := 16#0001 OR #Control_word; END_IF;
   IF NOT #CW_Off1_On THEN #Control_word := 16#FFFE AND #Control_word; END_IF;
END_REGION

REGION Network 3
   IF #CW_Off2 THEN #Control_word := 16#0002 OR #Control_word; END_IF;
   IF NOT #CW_Off2 THEN #Control_word := 16#FFFD AND #Control_word; END_IF;
END_REGION

REGION Network 4
   IF #CW_Off3 THEN #Control_word := 16#0004 OR #Control_word; END_IF;
   IF NOT #CW_Off3 THEN #Control_word := 16#FFFB AND #Control_word; END_IF;
END_REGION

REGION Network 5
   IF #CW_enable_operation THEN #Control_word := 16#0008 OR #Control_word; END_IF;
   IF NOT #CW_enable_operation THEN #Control_word := 16#FFF7 AND #Control_word; END_IF;
END_REGION

REGION Network 6
   IF #CW_no_lock_RFG THEN #Control_word := 16#0010 OR #Control_word; END_IF;
   IF NOT #CW_no_lock_RFG THEN #Control_word := 16#FFEF AND #Control_word; END_IF;
END_REGION

REGION Network 7
   IF #CW_no_stop_RFG THEN #Control_word := 16#0020 OR #Control_word; END_IF;
   IF NOT #CW_no_stop_RFG THEN #Control_word := 16#FFDF AND #Control_word; END_IF;
END_REGION

REGION Network 8
   IF #CW_enable_setpoint THEN #Control_word := 16#0040 OR #Control_word; END_IF;
   IF NOT #CW_enable_setpoint THEN #Control_word := 16#FFBF AND #Control_word; END_IF;
END_REGION

REGION Network 9
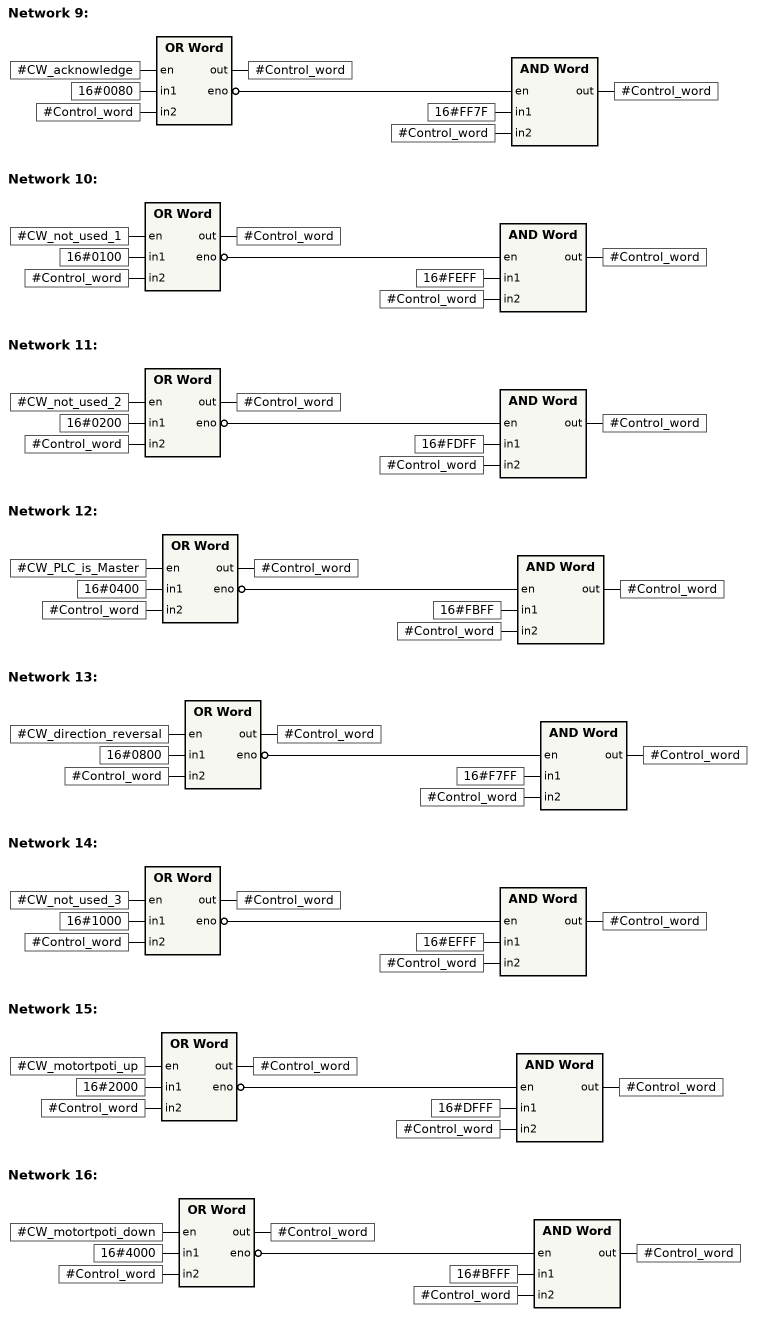
   IF #CW_acknowledge THEN #Control_word := 16#0080 OR #Control_word; END_IF;
   IF NOT #CW_acknowledge THEN #Control_word := 16#FF7F AND #Control_word; END_IF;
END_REGION

REGION Network 10
   IF #CW_not_used_1 THEN #Control_word := 16#0100 OR #Control_word; END_IF;
   IF NOT #CW_not_used_1 THEN #Control_word := 16#FEFF AND #Control_word; END_IF;
END_REGION

REGION Network 11
   IF #CW_not_used_2 THEN #Control_word := 16#0200 OR #Control_word; END_IF;
   IF NOT #CW_not_used_2 THEN #Control_word := 16#FDFF AND #Control_word; END_IF;
END_REGION

REGION Network 12
   IF #CW_PLC_is_Master THEN #Control_word := 16#0400 OR #Control_word; END_IF;
   IF NOT #CW_PLC_is_Master THEN #Control_word := 16#FBFF AND #Control_word; END_IF;
END_REGION

REGION Network 13
   IF #CW_direction_reversal THEN #Control_word := 16#0800 OR #Control_word; END_IF;
   IF NOT #CW_direction_reversal THEN #Control_word := 16#F7FF AND #Control_word; END_IF;
END_REGION

REGION Network 14
   IF #CW_not_used_3 THEN #Control_word := 16#1000 OR #Control_word; END_IF;
   IF NOT #CW_not_used_3 THEN #Control_word := 16#EFFF AND #Control_word; END_IF;
END_REGION

REGION Network 15
   IF #CW_motortpoti_up THEN #Control_word := 16#2000 OR #Control_word; END_IF;
   IF NOT #CW_motortpoti_up THEN #Control_word := 16#DFFF AND #Control_word; END_IF;
END_REGION

REGION Network 16
   IF #CW_motortpoti_down THEN #Control_word := 16#4000 OR #Control_word; END_IF;
   IF NOT #CW_motortpoti_down THEN #Control_word := 16#BFFF AND #Control_word; END_IF;
END_REGION

REGION Network 17
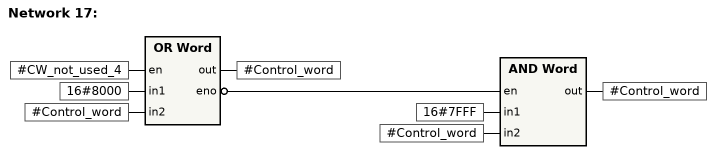
   IF #CW_not_used_4 THEN #Control_word := 16#8000 OR #Control_word; END_IF;
   IF NOT #CW_not_used_4 THEN #Control_word := 16#7FFF AND #Control_word; END_IF;
END_REGION
END_FUNCTION

FUNCTION_BLOCK "Inverter_Process_Data"   // FB1, FBD
{ S7_Optimized_Access := 'TRUE' }
VERSION : 0.1
// stored: AutoNumber false, IsIECCheckEnabled false, IsRetainMemResEnabled false, MemoryReserve 100, SetENOAutomatically false, UDAEnableTagReadback false
   VAR_INPUT
      control_word : Word := 16#0000;
      setpoint : Real;
      RD_address : HW_SUBMODULE;
      WR_address : HW_SUBMODULE;
      ref_quantity : Struct
         speed_p2000 : Real := 1500.0;
         current_p2002 : Real := 0.65;
         torque_p2003 : Real := 1.7;
      END_STRUCT;
   END_VAR
   VAR_OUTPUT
      status_word : Word;
      actual_speed : Real;
      actual_current : Real;
      actual_torque : Real;
      actual_alarm : Word;
      actual_fault : Word;
      RETVAL_RD : Word;
      RETVAL_WR : Word;
   END_VAR
   VAR_TEMP
      InData : Array[1..6] of Word;
      OutData : Array[1..6] of Word;
      actual_speed_INT : Int;
      actual_current_INT : Int;
      actual_torque_INT : Int;
      setpoint_INT : Int;
   END_VAR
BEGIN

REGION Network 1
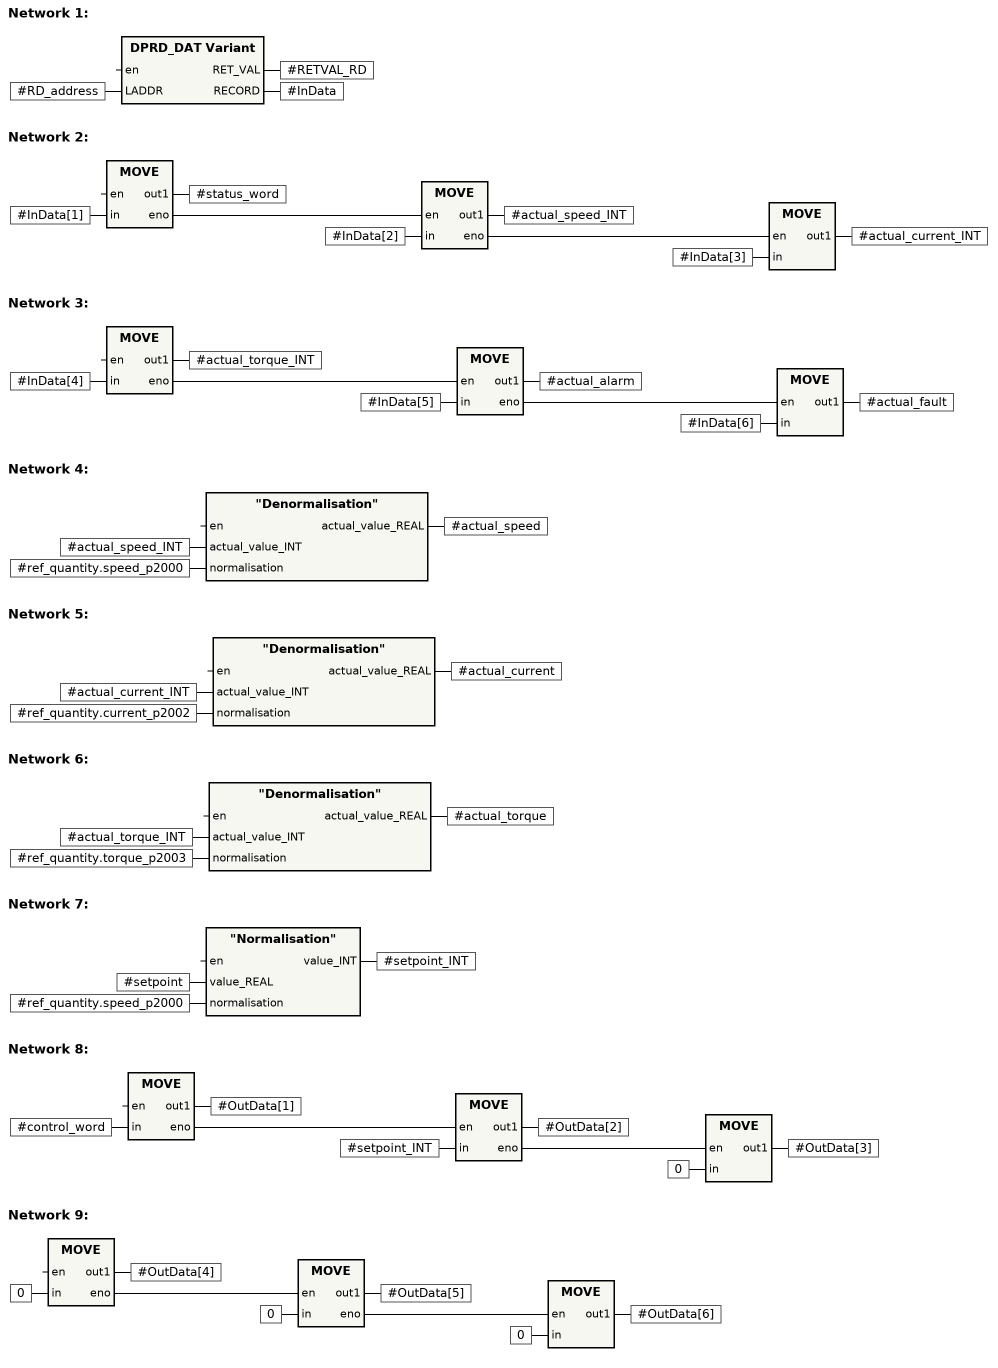
   #RETVAL_RD := DPRD_DAT(LADDR := #RD_address, RECORD => #InData);
END_REGION

REGION Network 2
   // ENO of a box is taken as its EN; it also drops when the box reports an error
   #status_word := #InData[1];
   #actual_speed_INT := #InData[2];
   #actual_current_INT := #InData[3];
END_REGION

REGION Network 3
   // ENO of a box is taken as its EN; it also drops when the box reports an error
   #actual_torque_INT := #InData[4];
   #actual_alarm := #InData[5];
   #actual_fault := #InData[6];
END_REGION

REGION Network 4
   "Denormalisation"(actual_value_INT := #actual_speed_INT,
                     normalisation := #ref_quantity.speed_p2000,
                     actual_value_REAL => #actual_speed);
END_REGION

REGION Network 5
   "Denormalisation"(actual_value_INT := #actual_current_INT,
                     normalisation := #ref_quantity.current_p2002,
                     actual_value_REAL => #actual_current);
END_REGION

REGION Network 6
   "Denormalisation"(actual_value_INT := #actual_torque_INT,
                     normalisation := #ref_quantity.torque_p2003,
                     actual_value_REAL => #actual_torque);
END_REGION

REGION Network 7
   "Normalisation"(value_REAL := #setpoint,
                   normalisation := #ref_quantity.speed_p2000,
                   value_INT => #setpoint_INT);
END_REGION

REGION Network 8
   // ENO of a box is taken as its EN; it also drops when the box reports an error
   #OutData[1] := #control_word;
   #OutData[2] := #setpoint_INT;
   #OutData[3] := 0;
END_REGION

REGION Network 9
   // ENO of a box is taken as its EN; it also drops when the box reports an error
   #OutData[4] := 0;
   #OutData[5] := 0;
   #OutData[6] := 0;
END_REGION

REGION Network 10
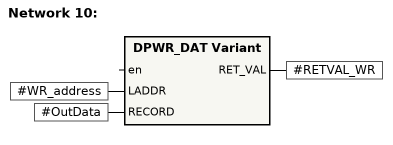
   #RETVAL_WR := DPWR_DAT(LADDR := #WR_address, RECORD := #OutData);
END_REGION
END_FUNCTION_BLOCK

FUNCTION "FC09_NoPressurePlate" : Void   // FC9, LAD
TITLE = Pressure palte isn't present
{ S7_Optimized_Access := 'FALSE' }
AUTHOR : Robopac
VERSION : 0.0
// stored: AutoNumber false, IsIECCheckEnabled false, SetENOAutomatically false, UDAEnableTagReadback false
BEGIN

REGION Network 1: Pressure plate bits
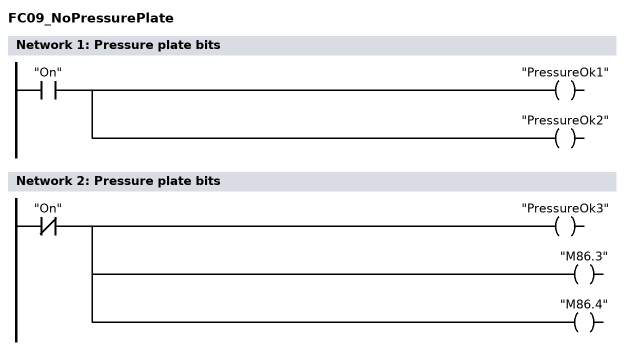
   RUNG wire#powerrail
      Contact( "On" )
      wire#w1
      Coil( "PressureOk1" )
   END_RUNG
   RUNG wire#w1
      Coil( "PressureOk2" )
   END_RUNG
   // the same network as SCL:
   "PressureOk1" := "On";
   "PressureOk2" := "On";
END_REGION

REGION Network 2: Pressure plate bits
   RUNG wire#powerrail
      I_Contact( "On" )
      wire#w1
      Coil( "PressureOk3" )
   END_RUNG
   RUNG wire#w1
      Coil( "M86.3" )
   END_RUNG
   RUNG wire#w1
      Coil( "M86.4" )
   END_RUNG
   // the same network as SCL:
   "PressureOk3" := NOT "On";
   "M86.3" := NOT "On";
   "M86.4" := NOT "On";
END_REGION
END_FUNCTION

FUNCTION "FC10_PressureCircularPn5W" : Void   // FC10, LAD
{ S7_Optimized_Access := 'FALSE' }
VERSION : 0.1
// stored: AutoNumber false, IsIECCheckEnabled false, SetENOAutomatically false, UDAEnableTagReadback false
   VAR_TEMP
      PressurePTime : Word;
   END_VAR
   VAR_TEMP   // added for the SCL form of the ladder/FBD networks
      _w1 : Bool;
   END_VAR
BEGIN

REGION Network 1
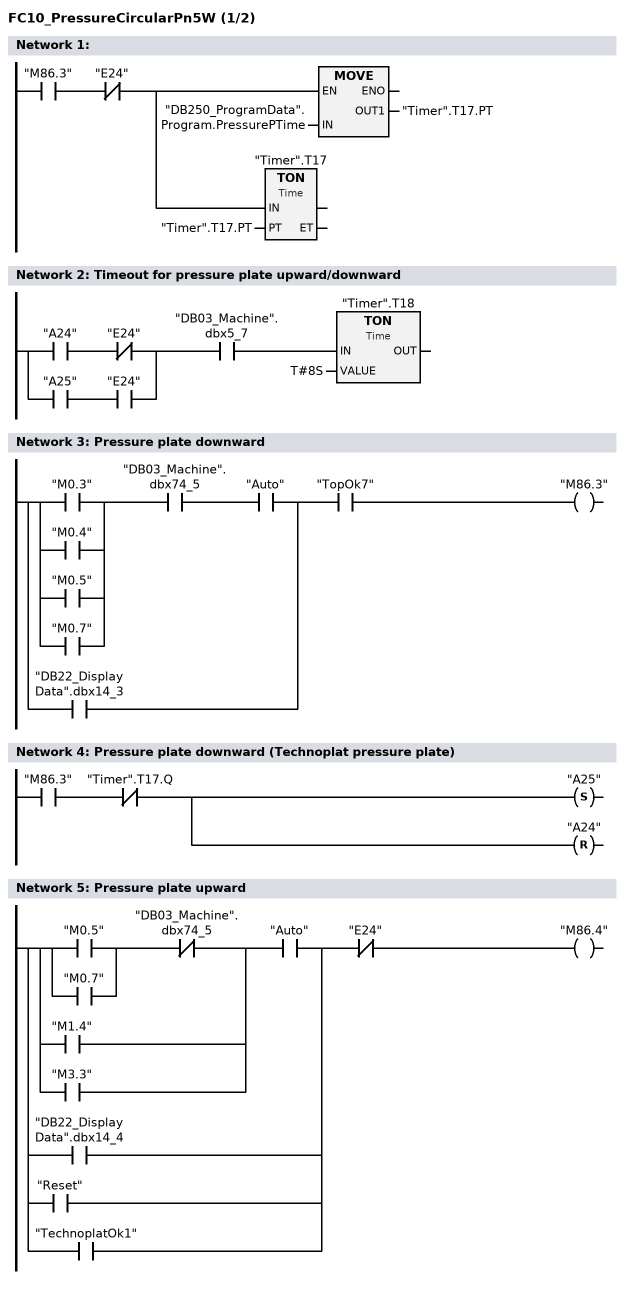
   RUNG wire#powerrail
      Contact( "M86.3" )
      I_Contact( "E24" )
      wire#w1
      { S7_GenerateENO := "TRUE" } Move(in := "DB250_ProgramData".Program.PressurePTime, out1 => "Timer".T17.PT)
   END_RUNG
   RUNG wire#w1
      { S7_Templates := "time_type := Time" } "Timer".T17.TON(pt := "Timer".T17.PT, et =>)
   END_RUNG
   // the same network as SCL:
   #_w1 := "M86.3" AND NOT "E24";
   IF #_w1 THEN "Timer".T17.PT := "DB250_ProgramData".Program.PressurePTime; END_IF;
   "Timer".T17.TON(IN := #_w1, PT := "Timer".T17.PT);
END_REGION

REGION Network 2: Timeout for pressure plate upward/downward
   "Timer".T18.TON(IN := (("A24" AND NOT "E24") OR ("A25" AND "E24")) AND "DB03_Machine".dbx5_7, PT := T#8S);   // TON coil
END_REGION

REGION Network 3: Pressure plate downward
   RUNG wire#powerrail
      Contact( "M0.3" )
      wire#w1
      Contact( "DB03_Machine".dbx74_5 )
      Contact( "Auto" )
      wire#w2
      Contact( "TopOk7" )
      Coil( "M86.3" )
   END_RUNG
   RUNG wire#powerrail
      Contact( "M0.4" )
   END_RUNG wire#w1
   RUNG wire#powerrail
      Contact( "M0.5" )
   END_RUNG wire#w1
   RUNG wire#powerrail
      Contact( "M0.7" )
   END_RUNG wire#w1
   RUNG wire#powerrail
      Contact( "DB22_DisplayData".dbx14_3 )
   END_RUNG wire#w2
   // the same network as SCL:
   "M86.3" := ((("M0.3" OR "M0.4" OR "M0.5" OR "M0.7") AND "DB03_Machine".dbx74_5 AND "Auto") OR "DB22_DisplayData".dbx14_3) AND "TopOk7";
END_REGION

REGION Network 4: Pressure plate downward (Technoplat pressure plate)
   RUNG wire#powerrail
      Contact( "M86.3" )
      I_Contact( "Timer".T17.Q )
      wire#w1
      S_Coil( "A25" )
   END_RUNG
   RUNG wire#w1
      R_Coil( "A24" )
   END_RUNG
   // the same network as SCL:
   IF "M86.3" AND NOT "Timer".T17.Q THEN
       "A25" := TRUE;
       "A24" := FALSE;
   END_IF;
END_REGION

REGION Network 5: Pressure plate upward
   RUNG wire#powerrail
      Contact( "M0.5" )
      wire#w1
      I_Contact( "DB03_Machine".dbx74_5 )
      wire#w2
      Contact( "Auto" )
      wire#w3
      I_Contact( "E24" )
      Coil( "M86.4" )
   END_RUNG
   RUNG wire#powerrail
      Contact( "M0.7" )
   END_RUNG wire#w1
   RUNG wire#powerrail
      Contact( "M1.4" )
   END_RUNG wire#w2
   RUNG wire#powerrail
      Contact( "M3.3" )
   END_RUNG wire#w2
   RUNG wire#powerrail
      Contact( "DB22_DisplayData".dbx14_4 )
   END_RUNG wire#w3
   RUNG wire#powerrail
      Contact( "Reset" )
   END_RUNG wire#w3
   RUNG wire#powerrail
      Contact( "TechnoplatOk1" )
   END_RUNG wire#w3
   // the same network as SCL:
   "M86.4" := ((((("M0.5" OR "M0.7") AND NOT "DB03_Machine".dbx74_5) OR "M1.4" OR "M3.3") AND "Auto") OR "DB22_DisplayData".dbx14_4 OR "Reset" OR "TechnoplatOk1") AND NOT "E24";
END_REGION

REGION Network 6: Pressure plate upward (Technoplat pressure plate)
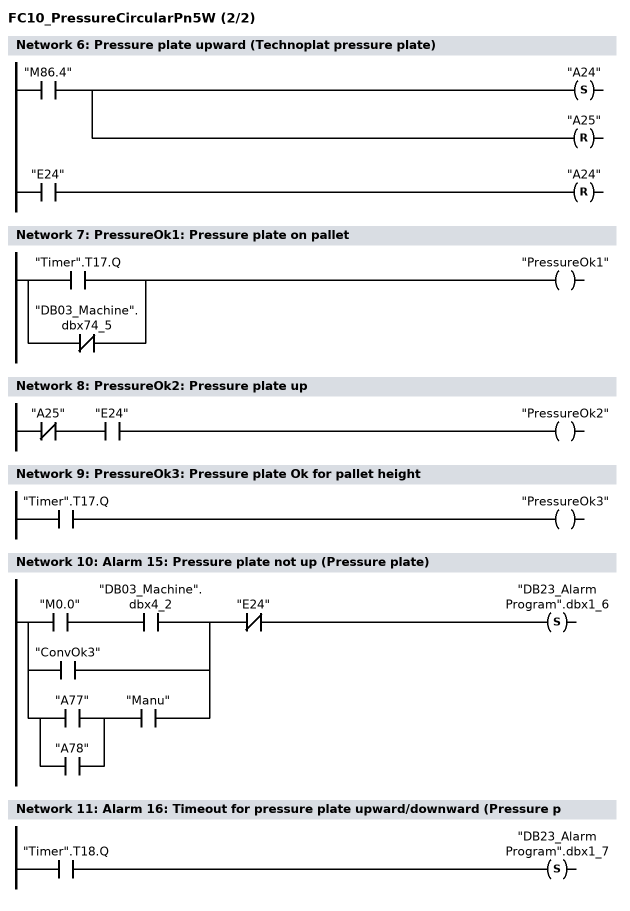
   RUNG wire#powerrail
      Contact( "M86.4" )
      wire#w1
      S_Coil( "A24" )
   END_RUNG
   RUNG wire#w1
      R_Coil( "A25" )
   END_RUNG
   RUNG wire#powerrail
      Contact( "E24" )
      R_Coil( "A24" )
   END_RUNG
   // the same network as SCL:
   IF "M86.4" THEN
       "A24" := TRUE;
       "A25" := FALSE;
   END_IF;
   IF "E24" THEN "A24" := FALSE; END_IF;
END_REGION

REGION Network 7: PressureOk1: Pressure plate on pallet
   RUNG wire#powerrail
      Contact( "Timer".T17.Q )
      wire#w1
      Coil( "PressureOk1" )
   END_RUNG
   RUNG wire#powerrail
      I_Contact( "DB03_Machine".dbx74_5 )
   END_RUNG wire#w1
   // the same network as SCL:
   "PressureOk1" := "Timer".T17.Q OR NOT "DB03_Machine".dbx74_5;
END_REGION

REGION Network 8: PressureOk2: Pressure plate up
   RUNG wire#powerrail
      I_Contact( "A25" )
      Contact( "E24" )
      Coil( "PressureOk2" )
   END_RUNG
   // the same network as SCL:
   "PressureOk2" := NOT "A25" AND "E24";
END_REGION

REGION Network 9: PressureOk3: Pressure plate Ok for pallet height
   RUNG wire#powerrail
      Contact( "Timer".T17.Q )
      Coil( "PressureOk3" )
   END_RUNG
   // the same network as SCL:
   "PressureOk3" := "Timer".T17.Q;
END_REGION

REGION Network 10: Alarm 15: Pressure plate not up (Pressure plate)
   RUNG wire#powerrail
      Contact( "M0.0" )
      Contact( "DB03_Machine".dbx4_2 )
      wire#w1
      I_Contact( "E24" )
      S_Coil( "DB23_AlarmProgram".dbx1_6 )
   END_RUNG
   RUNG wire#powerrail
      Contact( "ConvOk3" )
   END_RUNG wire#w1
   RUNG wire#powerrail
      Contact( "A77" )
      wire#w2
      Contact( "Manu" )
   END_RUNG wire#w1
   RUNG wire#powerrail
      Contact( "A78" )
   END_RUNG wire#w2
   // the same network as SCL:
   IF (("M0.0" AND "DB03_Machine".dbx4_2) OR "ConvOk3" OR (("A77" OR "A78") AND "Manu")) AND NOT "E24" THEN
       "DB23_AlarmProgram".dbx1_6 := TRUE;
   END_IF;
END_REGION

REGION Network 11: Alarm 16: Timeout for pressure plate upward/downward (Pressure p
   RUNG wire#powerrail
      Contact( "Timer".T18.Q )
      S_Coil( "DB23_AlarmProgram".dbx1_7 )
   END_RUNG
   // the same network as SCL:
   IF "Timer".T18.Q THEN "DB23_AlarmProgram".dbx1_7 := TRUE; END_IF;
END_REGION
END_FUNCTION

FUNCTION "FC12_PressureCircularMono" : Void   // FC12, LAD
{ S7_Optimized_Access := 'FALSE' }
VERSION : 0.1
// stored: AutoNumber false, IsIECCheckEnabled false, SetENOAutomatically false, UDAEnableTagReadback false
   VAR_TEMP
      PressurePTime : Word;
   END_VAR
   VAR_TEMP   // added for the SCL form of the ladder/FBD networks
      _w1 : Bool;
   END_VAR
BEGIN

REGION Network 1
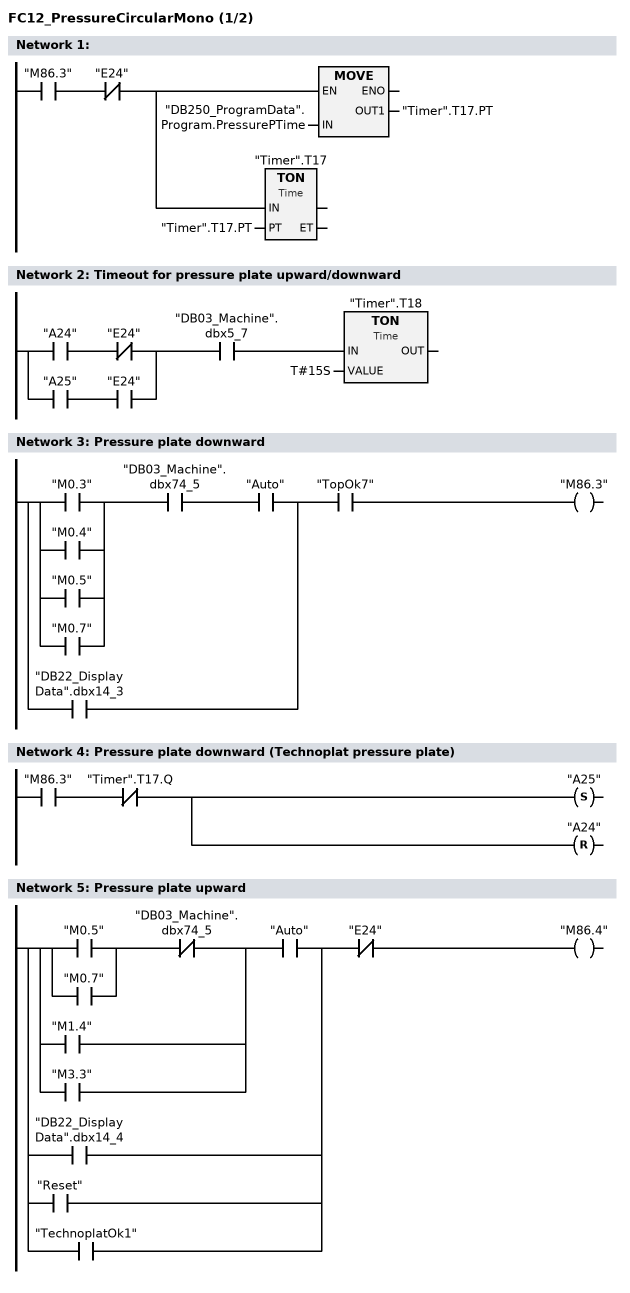
   RUNG wire#powerrail
      Contact( "M86.3" )
      I_Contact( "E24" )
      wire#w1
      { S7_GenerateENO := "TRUE" } Move(in := "DB250_ProgramData".Program.PressurePTime, out1 => "Timer".T17.PT)
   END_RUNG
   RUNG wire#w1
      { S7_Templates := "time_type := Time" } "Timer".T17.TON(pt := "Timer".T17.PT, et =>)
   END_RUNG
   // the same network as SCL:
   #_w1 := "M86.3" AND NOT "E24";
   IF #_w1 THEN "Timer".T17.PT := "DB250_ProgramData".Program.PressurePTime; END_IF;
   "Timer".T17.TON(IN := #_w1, PT := "Timer".T17.PT);
END_REGION

REGION Network 2: Timeout for pressure plate upward/downward
   "Timer".T18.TON(IN := (("A24" AND NOT "E24") OR ("A25" AND "E24")) AND "DB03_Machine".dbx5_7, PT := T#15S);   // TON coil
END_REGION

REGION Network 3: Pressure plate downward
   RUNG wire#powerrail
      Contact( "M0.3" )
      wire#w1
      Contact( "DB03_Machine".dbx74_5 )
      Contact( "Auto" )
      wire#w2
      Contact( "TopOk7" )
      Coil( "M86.3" )
   END_RUNG
   RUNG wire#powerrail
      Contact( "M0.4" )
   END_RUNG wire#w1
   RUNG wire#powerrail
      Contact( "M0.5" )
   END_RUNG wire#w1
   RUNG wire#powerrail
      Contact( "M0.7" )
   END_RUNG wire#w1
   RUNG wire#powerrail
      Contact( "DB22_DisplayData".dbx14_3 )
   END_RUNG wire#w2
   // the same network as SCL:
   "M86.3" := ((("M0.3" OR "M0.4" OR "M0.5" OR "M0.7") AND "DB03_Machine".dbx74_5 AND "Auto") OR "DB22_DisplayData".dbx14_3) AND "TopOk7";
END_REGION

REGION Network 4: Pressure plate downward (Technoplat pressure plate)
   RUNG wire#powerrail
      Contact( "M86.3" )
      I_Contact( "Timer".T17.Q )
      wire#w1
      S_Coil( "A25" )
   END_RUNG
   RUNG wire#w1
      R_Coil( "A24" )
   END_RUNG
   // the same network as SCL:
   IF "M86.3" AND NOT "Timer".T17.Q THEN
       "A25" := TRUE;
       "A24" := FALSE;
   END_IF;
END_REGION

REGION Network 5: Pressure plate upward
   RUNG wire#powerrail
      Contact( "M0.5" )
      wire#w1
      I_Contact( "DB03_Machine".dbx74_5 )
      wire#w2
      Contact( "Auto" )
      wire#w3
      I_Contact( "E24" )
      Coil( "M86.4" )
   END_RUNG
   RUNG wire#powerrail
      Contact( "M0.7" )
   END_RUNG wire#w1
   RUNG wire#powerrail
      Contact( "M1.4" )
   END_RUNG wire#w2
   RUNG wire#powerrail
      Contact( "M3.3" )
   END_RUNG wire#w2
   RUNG wire#powerrail
      Contact( "DB22_DisplayData".dbx14_4 )
   END_RUNG wire#w3
   RUNG wire#powerrail
      Contact( "Reset" )
   END_RUNG wire#w3
   RUNG wire#powerrail
      Contact( "TechnoplatOk1" )
   END_RUNG wire#w3
   // the same network as SCL:
   "M86.4" := ((((("M0.5" OR "M0.7") AND NOT "DB03_Machine".dbx74_5) OR "M1.4" OR "M3.3") AND "Auto") OR "DB22_DisplayData".dbx14_4 OR "Reset" OR "TechnoplatOk1") AND NOT "E24";
END_REGION

REGION Network 6: Pressure plate upward (Technoplat pressure plate)
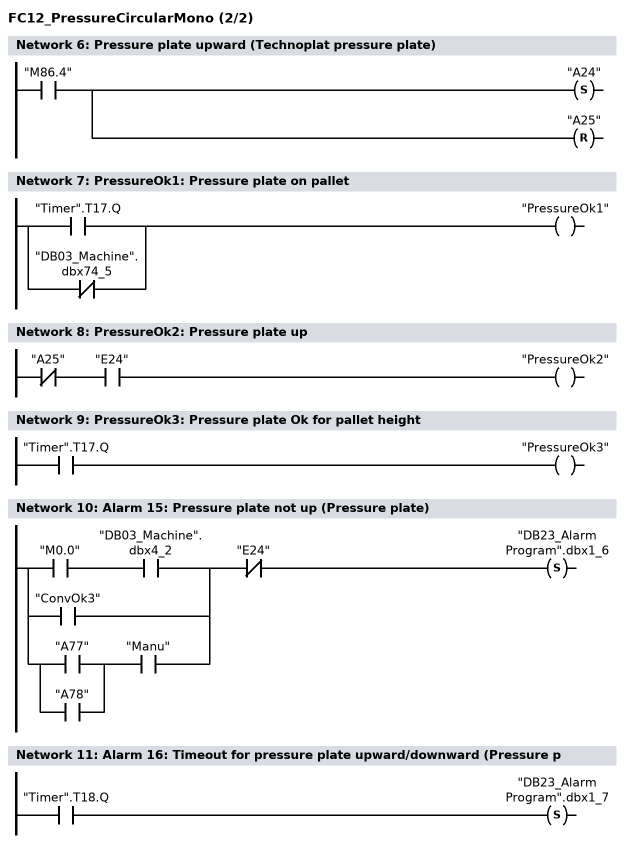
   RUNG wire#powerrail
      Contact( "M86.4" )
      wire#w1
      S_Coil( "A24" )
   END_RUNG
   RUNG wire#w1
      R_Coil( "A25" )
   END_RUNG
   // the same network as SCL:
   IF "M86.4" THEN
       "A24" := TRUE;
       "A25" := FALSE;
   END_IF;
END_REGION

REGION Network 7: PressureOk1: Pressure plate on pallet
   RUNG wire#powerrail
      Contact( "Timer".T17.Q )
      wire#w1
      Coil( "PressureOk1" )
   END_RUNG
   RUNG wire#powerrail
      I_Contact( "DB03_Machine".dbx74_5 )
   END_RUNG wire#w1
   // the same network as SCL:
   "PressureOk1" := "Timer".T17.Q OR NOT "DB03_Machine".dbx74_5;
END_REGION

REGION Network 8: PressureOk2: Pressure plate up
   RUNG wire#powerrail
      I_Contact( "A25" )
      Contact( "E24" )
      Coil( "PressureOk2" )
   END_RUNG
   // the same network as SCL:
   "PressureOk2" := NOT "A25" AND "E24";
END_REGION

REGION Network 9: PressureOk3: Pressure plate Ok for pallet height
   RUNG wire#powerrail
      Contact( "Timer".T17.Q )
      Coil( "PressureOk3" )
   END_RUNG
   // the same network as SCL:
   "PressureOk3" := "Timer".T17.Q;
END_REGION

REGION Network 10: Alarm 15: Pressure plate not up (Pressure plate)
   RUNG wire#powerrail
      Contact( "M0.0" )
      Contact( "DB03_Machine".dbx4_2 )
      wire#w1
      I_Contact( "E24" )
      S_Coil( "DB23_AlarmProgram".dbx1_6 )
   END_RUNG
   RUNG wire#powerrail
      Contact( "ConvOk3" )
   END_RUNG wire#w1
   RUNG wire#powerrail
      Contact( "A77" )
      wire#w2
      Contact( "Manu" )
   END_RUNG wire#w1
   RUNG wire#powerrail
      Contact( "A78" )
   END_RUNG wire#w2
   // the same network as SCL:
   IF (("M0.0" AND "DB03_Machine".dbx4_2) OR "ConvOk3" OR (("A77" OR "A78") AND "Manu")) AND NOT "E24" THEN
       "DB23_AlarmProgram".dbx1_6 := TRUE;
   END_IF;
END_REGION

REGION Network 11: Alarm 16: Timeout for pressure plate upward/downward (Pressure p
   RUNG wire#powerrail
      Contact( "Timer".T18.Q )
      S_Coil( "DB23_AlarmProgram".dbx1_7 )
   END_RUNG
   // the same network as SCL:
   IF "Timer".T18.Q THEN "DB23_AlarmProgram".dbx1_7 := TRUE; END_IF;
END_REGION
END_FUNCTION

FUNCTION "FC26_Pos1SensorDec" : Void   // FC26, LAD
{ S7_Optimized_Access := 'FALSE' }
VERSION : 0.1
// stored: AutoNumber false, IsIECCheckEnabled false, SetENOAutomatically false, UDAEnableTagReadback false
BEGIN

REGION Network 1: Delay on pallet positioning
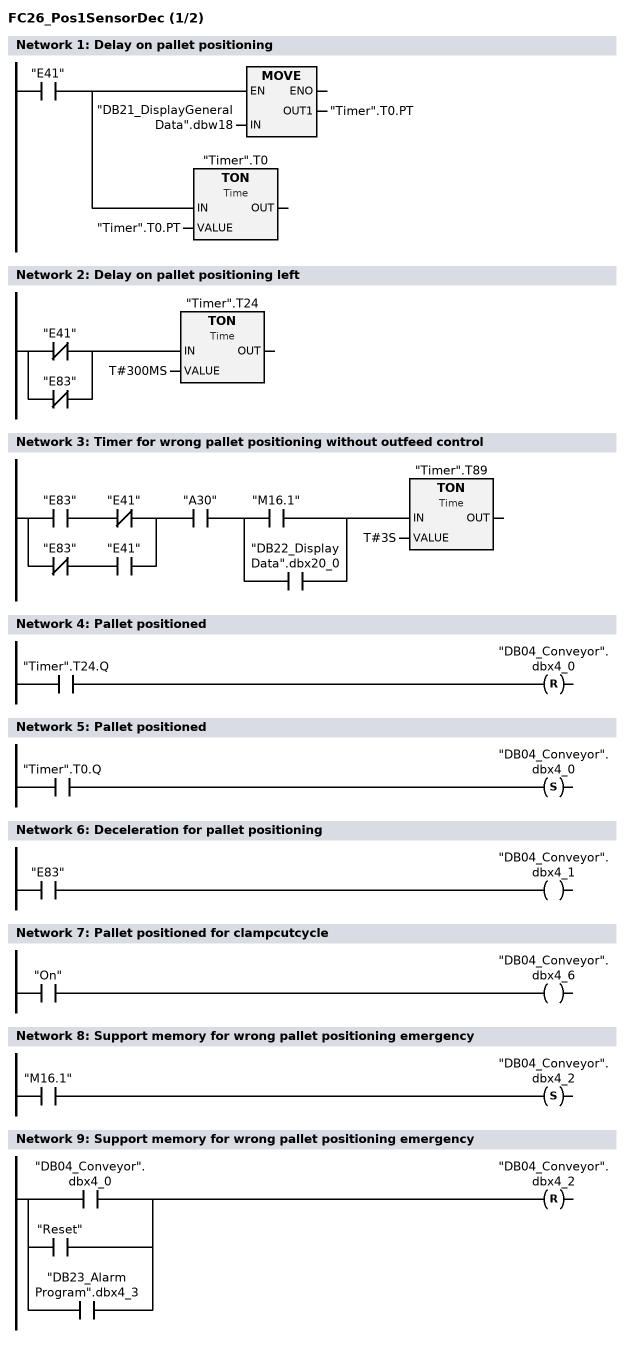
   IF "E41" THEN "Timer".T0.PT := "DB21_DisplayGeneralData".dbw18; END_IF;
   "Timer".T0.TON(IN := "E41", PT := "Timer".T0.PT);   // TON coil
END_REGION

REGION Network 2: Delay on pallet positioning left
   "Timer".T24.TON(IN := NOT "E41" OR NOT "E83", PT := T#300MS);   // TON coil
END_REGION

REGION Network 3: Timer for wrong pallet positioning without outfeed control
   "Timer".T89.TON(IN := (("E83" AND NOT "E41") OR (NOT "E83" AND "E41")) AND "A30" AND ("M16.1" OR "DB22_DisplayData".dbx20_0), PT := T#3S);   // TON coil
END_REGION

REGION Network 4: Pallet positioned
   RUNG wire#powerrail
      Contact( "Timer".T24.Q )
      R_Coil( "DB04_Conveyor".dbx4_0 )
   END_RUNG
   // the same network as SCL:
   IF "Timer".T24.Q THEN "DB04_Conveyor".dbx4_0 := FALSE; END_IF;
END_REGION

REGION Network 5: Pallet positioned
   RUNG wire#powerrail
      Contact( "Timer".T0.Q )
      S_Coil( "DB04_Conveyor".dbx4_0 )
   END_RUNG
   // the same network as SCL:
   IF "Timer".T0.Q THEN "DB04_Conveyor".dbx4_0 := TRUE; END_IF;
END_REGION

REGION Network 6: Deceleration for pallet positioning
   RUNG wire#powerrail
      Contact( "E83" )
      Coil( "DB04_Conveyor".dbx4_1 )
   END_RUNG
   // the same network as SCL:
   "DB04_Conveyor".dbx4_1 := "E83";
END_REGION

REGION Network 7: Pallet positioned for clampcutcycle
   RUNG wire#powerrail
      Contact( "On" )
      Coil( "DB04_Conveyor".dbx4_6 )
   END_RUNG
   // the same network as SCL:
   "DB04_Conveyor".dbx4_6 := "On";
END_REGION

REGION Network 8: Support memory for wrong pallet positioning emergency
   RUNG wire#powerrail
      Contact( "M16.1" )
      S_Coil( "DB04_Conveyor".dbx4_2 )
   END_RUNG
   // the same network as SCL:
   IF "M16.1" THEN "DB04_Conveyor".dbx4_2 := TRUE; END_IF;
END_REGION

REGION Network 9: Support memory for wrong pallet positioning emergency
   RUNG wire#powerrail
      Contact( "DB04_Conveyor".dbx4_0 )
      wire#w1
      R_Coil( "DB04_Conveyor".dbx4_2 )
   END_RUNG
   RUNG wire#powerrail
      Contact( "Reset" )
   END_RUNG wire#w1
   RUNG wire#powerrail
      Contact( "DB23_AlarmProgram".dbx4_3 )
   END_RUNG wire#w1
   // the same network as SCL:
   IF "DB04_Conveyor".dbx4_0 OR "Reset" OR "DB23_AlarmProgram".dbx4_3 THEN
       "DB04_Conveyor".dbx4_2 := FALSE;
   END_IF;
END_REGION

REGION Network 10: Alarm 33: Pallet positioning released during table rotation (Con
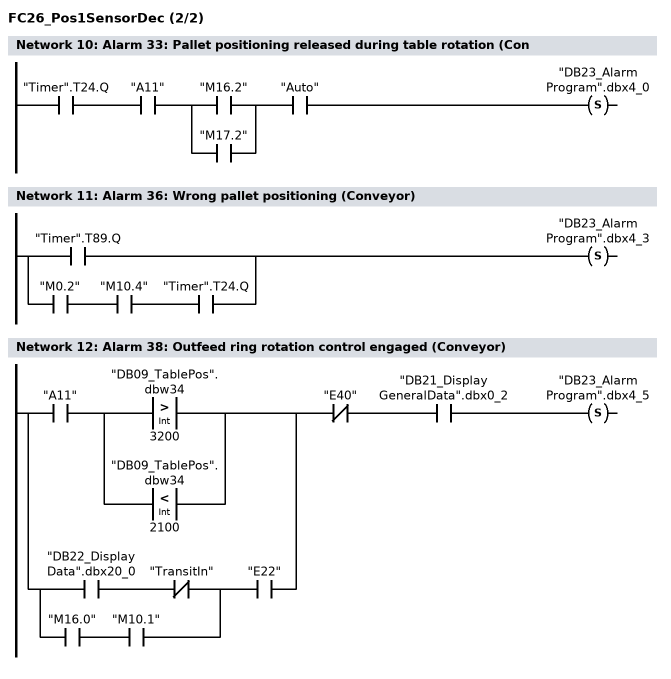
   RUNG wire#powerrail
      Contact( "Timer".T24.Q )
      Contact( "A11" )
      wire#w1
      Contact( "M16.2" )
      wire#w2
      Contact( "Auto" )
      S_Coil( "DB23_AlarmProgram".dbx4_0 )
   END_RUNG
   RUNG wire#w1
      Contact( "M17.2" )
   END_RUNG wire#w2
   // the same network as SCL:
   IF "Timer".T24.Q AND "A11" AND ("M16.2" OR "M17.2") AND "Auto" THEN
       "DB23_AlarmProgram".dbx4_0 := TRUE;
   END_IF;
END_REGION

REGION Network 11: Alarm 36: Wrong pallet positioning (Conveyor)
   RUNG wire#powerrail
      Contact( "Timer".T89.Q )
      wire#w1
      S_Coil( "DB23_AlarmProgram".dbx4_3 )
   END_RUNG
   RUNG wire#powerrail
      Contact( "M0.2" )
      Contact( "M10.4" )
      Contact( "Timer".T24.Q )
   END_RUNG wire#w1
   // the same network as SCL:
   IF "Timer".T89.Q OR ("M0.2" AND "M10.4" AND "Timer".T24.Q) THEN
       "DB23_AlarmProgram".dbx4_3 := TRUE;
   END_IF;
END_REGION

REGION Network 12: Alarm 38: Outfeed ring rotation control engaged (Conveyor)
   RUNG wire#powerrail
      Contact( "A11" )
      wire#w1
      { S7_Templates := "SrcType := Int" } GT_Contact(in1 := "DB09_TablePos".dbw34, in2 := 3200)
      wire#w2
      I_Contact( "E40" )
      Contact( "DB21_DisplayGeneralData".dbx0_2 )
      S_Coil( "DB23_AlarmProgram".dbx4_5 )
   END_RUNG
   RUNG wire#w1
      { S7_Templates := "SrcType := Int" } LT_Contact(in1 := "DB09_TablePos".dbw34, in2 := 2100)
   END_RUNG wire#w2
   RUNG wire#powerrail
      Contact( "DB22_DisplayData".dbx20_0 )
      I_Contact( "TransitIn" )
      wire#w3
      Contact( "E22" )
   END_RUNG wire#w2
   RUNG wire#powerrail
      Contact( "M16.0" )
      Contact( "M10.1" )
   END_RUNG wire#w3
   // the same network as SCL:
   IF (("A11" AND (("DB09_TablePos".dbw34 > 3200) OR ("DB09_TablePos".dbw34 < 2100))) OR ((("DB22_DisplayData".dbx20_0 AND NOT "TransitIn") OR ("M16.0" AND "M10.1")) AND "E22")) AND NOT "E40" AND "DB21_DisplayGeneralData".dbx0_2 THEN
       "DB23_AlarmProgram".dbx4_5 := TRUE;
   END_IF;
END_REGION
END_FUNCTION

FUNCTION "FC27_PosSelfcEncoder" : Void   // FC27, LAD
TITLE = Pallet positioning with selfcentering system and encoder
{ S7_Optimized_Access := 'FALSE' }
AUTHOR : Robopac
VERSION : 0.0
// stored: AutoNumber false, IsIECCheckEnabled false, SetENOAutomatically false, UDAEnableTagReadback false
   VAR_TEMP
      Ch7ValmmEnco1 : DInt;
      Ch7ValmmEnco2 : DInt;
      PalletLenghtdiv2 : Int;
      PosToReach : Int;
      PosToDecelation : Int;
      WTemp1 : Int;
      DWTemp1 : DInt;
      DWTemp2 : DInt;
   END_VAR
   VAR_TEMP   // added for the SCL form of the ladder/FBD networks
      _w1 : Bool;
      _w2 : Bool;
   END_VAR
BEGIN

REGION Network 1: Delay on pallet positioning left
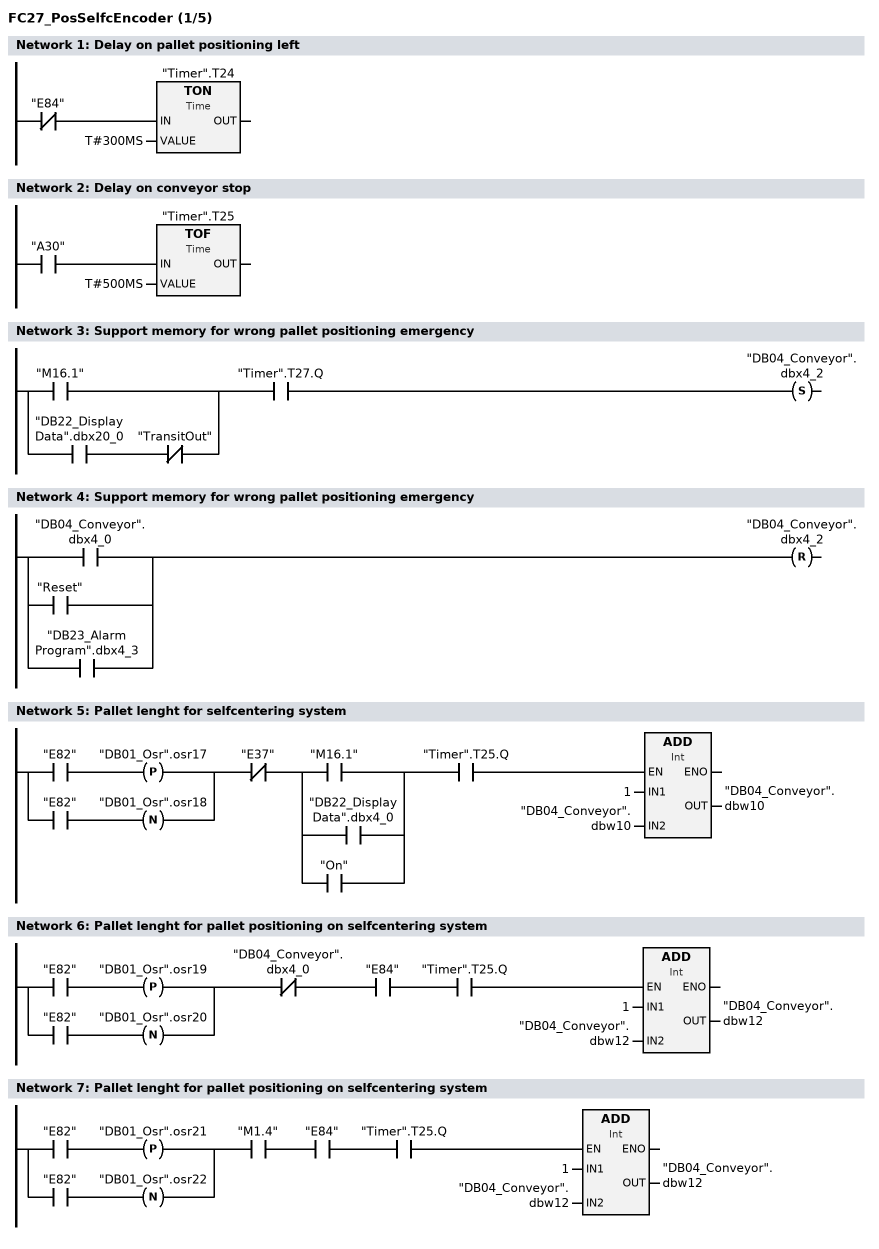
   "Timer".T24.TON(IN := NOT "E84", PT := T#300MS);   // TON coil
END_REGION

REGION Network 2: Delay on conveyor stop
   "Timer".T25.TOF(IN := "A30", PT := T#500MS);   // TOF coil
END_REGION

REGION Network 3: Support memory for wrong pallet positioning emergency
   RUNG wire#powerrail
      Contact( "M16.1" )
      wire#w1
      Contact( "Timer".T27.Q )
      S_Coil( "DB04_Conveyor".dbx4_2 )
   END_RUNG
   RUNG wire#powerrail
      Contact( "DB22_DisplayData".dbx20_0 )
      I_Contact( "TransitOut" )
   END_RUNG wire#w1
   // the same network as SCL:
   IF ("M16.1" OR ("DB22_DisplayData".dbx20_0 AND NOT "TransitOut")) AND "Timer".T27.Q THEN
       "DB04_Conveyor".dbx4_2 := TRUE;
   END_IF;
END_REGION

REGION Network 4: Support memory for wrong pallet positioning emergency
   RUNG wire#powerrail
      Contact( "DB04_Conveyor".dbx4_0 )
      wire#w1
      R_Coil( "DB04_Conveyor".dbx4_2 )
   END_RUNG
   RUNG wire#powerrail
      Contact( "Reset" )
   END_RUNG wire#w1
   RUNG wire#powerrail
      Contact( "DB23_AlarmProgram".dbx4_3 )
   END_RUNG wire#w1
   // the same network as SCL:
   IF "DB04_Conveyor".dbx4_0 OR "Reset" OR "DB23_AlarmProgram".dbx4_3 THEN
       "DB04_Conveyor".dbx4_2 := FALSE;
   END_IF;
END_REGION

REGION Network 5: Pallet lenght for selfcentering system
   RUNG wire#powerrail
      Contact( "E82" )
      P_Trig( "DB01_Osr".osr17 )
      wire#w1
      I_Contact( "E37" )
      wire#w2
      Contact( "M16.1" )
      wire#w3
      Contact( "Timer".T25.Q )
      { S7_Templates := "SrcType := Int"; S7_GenerateENO := "TRUE" } Add(in1 := 1, in2 := "DB04_Conveyor".dbw10, out => "DB04_Conveyor".dbw10)
   END_RUNG
   RUNG wire#powerrail
      Contact( "E82" )
      N_Trig( "DB01_Osr".osr18 )
   END_RUNG wire#w1
   RUNG wire#w2
      Contact( "DB22_DisplayData".dbx4_0 )
   END_RUNG wire#w3
   RUNG wire#w2
      Contact( "On" )
   END_RUNG wire#w3
   // the same network as SCL:
   #_w1 := "E82" AND NOT "DB01_Osr".osr17;   // rising edge
   "DB01_Osr".osr17 := "E82";
   #_w2 := NOT "E82" AND "DB01_Osr".osr18;   // falling edge
   "DB01_Osr".osr18 := "E82";
   IF (#_w1 OR #_w2) AND NOT "E37" AND ("M16.1" OR "DB22_DisplayData".dbx4_0 OR "On") AND "Timer".T25.Q THEN
       "DB04_Conveyor".dbw10 := 1 + "DB04_Conveyor".dbw10;
   END_IF;
END_REGION

REGION Network 6: Pallet lenght for pallet positioning on selfcentering system
   RUNG wire#powerrail
      Contact( "E82" )
      P_Trig( "DB01_Osr".osr19 )
      wire#w1
      I_Contact( "DB04_Conveyor".dbx4_0 )
      Contact( "E84" )
      Contact( "Timer".T25.Q )
      { S7_Templates := "SrcType := Int"; S7_GenerateENO := "TRUE" } Add(in1 := 1, in2 := "DB04_Conveyor".dbw12, out => "DB04_Conveyor".dbw12)
   END_RUNG
   RUNG wire#powerrail
      Contact( "E82" )
      N_Trig( "DB01_Osr".osr20 )
   END_RUNG wire#w1
   // the same network as SCL:
   #_w1 := "E82" AND NOT "DB01_Osr".osr19;   // rising edge
   "DB01_Osr".osr19 := "E82";
   #_w2 := NOT "E82" AND "DB01_Osr".osr20;   // falling edge
   "DB01_Osr".osr20 := "E82";
   IF (#_w1 OR #_w2) AND NOT "DB04_Conveyor".dbx4_0 AND "E84" AND "Timer".T25.Q THEN
       "DB04_Conveyor".dbw12 := 1 + "DB04_Conveyor".dbw12;
   END_IF;
END_REGION

REGION Network 7: Pallet lenght for pallet positioning on selfcentering system
   RUNG wire#powerrail
      Contact( "E82" )
      P_Trig( "DB01_Osr".osr21 )
      wire#w1
      Contact( "M1.4" )
      Contact( "E84" )
      Contact( "Timer".T25.Q )
      { S7_Templates := "SrcType := Int"; S7_GenerateENO := "TRUE" } Add(in1 := 1, in2 := "DB04_Conveyor".dbw12, out => "DB04_Conveyor".dbw12)
   END_RUNG
   RUNG wire#powerrail
      Contact( "E82" )
      N_Trig( "DB01_Osr".osr22 )
   END_RUNG wire#w1
   // the same network as SCL:
   #_w1 := "E82" AND NOT "DB01_Osr".osr21;   // rising edge
   "DB01_Osr".osr21 := "E82";
   #_w2 := NOT "E82" AND "DB01_Osr".osr22;   // falling edge
   "DB01_Osr".osr22 := "E82";
   IF (#_w1 OR #_w2) AND "M1.4" AND "E84" AND "Timer".T25.Q THEN
       "DB04_Conveyor".dbw12 := 1 + "DB04_Conveyor".dbw12;
   END_IF;
END_REGION

REGION Network 8: Reset pallet lenght
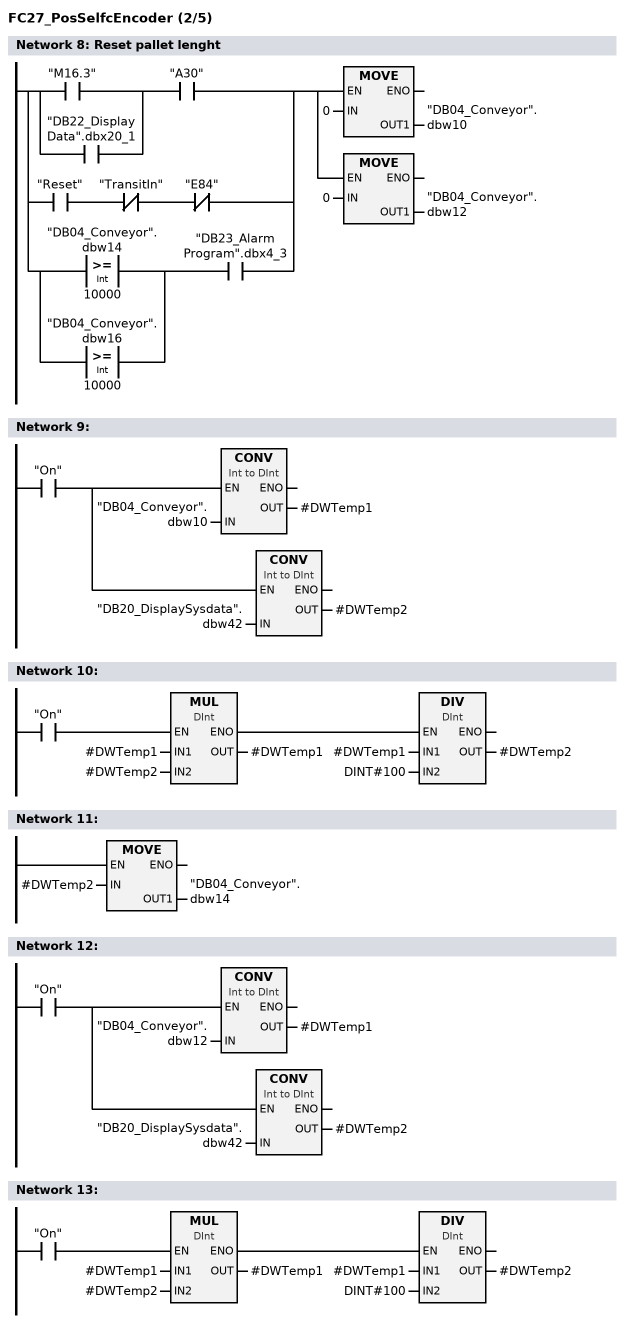
   RUNG wire#powerrail
      Contact( "M16.3" )
      wire#w1
      Contact( "A30" )
      wire#w2
      { S7_GenerateENO := "TRUE" } Move(in := 0, out1 => "DB04_Conveyor".dbw10)
   END_RUNG
   RUNG wire#powerrail
      Contact( "DB22_DisplayData".dbx20_1 )
   END_RUNG wire#w1
   RUNG wire#powerrail
      Contact( "Reset" )
      I_Contact( "TransitIn" )
      I_Contact( "E84" )
   END_RUNG wire#w2
   RUNG wire#powerrail
      { S7_Templates := "SrcType := Int" } GE_Contact(in1 := "DB04_Conveyor".dbw14, in2 := 10000)
      wire#w3
      Contact( "DB23_AlarmProgram".dbx4_3 )
   END_RUNG wire#w2
   RUNG wire#powerrail
      { S7_Templates := "SrcType := Int" } GE_Contact(in1 := "DB04_Conveyor".dbw16, in2 := 10000)
   END_RUNG wire#w3
   RUNG wire#w2
      { S7_GenerateENO := "TRUE" } Move(in := 0, out1 => "DB04_Conveyor".dbw12)
   END_RUNG
   // the same network as SCL:
   IF (("M16.3" OR "DB22_DisplayData".dbx20_1) AND "A30") OR ("Reset" AND NOT "TransitIn" AND NOT "E84") OR ((("DB04_Conveyor".dbw14 >= 10000) OR ("DB04_Conveyor".dbw16 >= 10000)) AND "DB23_AlarmProgram".dbx4_3) THEN
       "DB04_Conveyor".dbw10 := 0;
       "DB04_Conveyor".dbw12 := 0;
   END_IF;
END_REGION

REGION Network 9
   RUNG wire#powerrail
      Contact( "On" )
      wire#w1
      { S7_Templates := "[SrcType := Int, DestType := DInt]"; S7_GenerateENO := "TRUE" } Convert(in := "DB04_Conveyor".dbw10, out => #DWTemp1)
   END_RUNG
   RUNG wire#w1
      { S7_Templates := "[SrcType := Int, DestType := DInt]"; S7_GenerateENO := "TRUE" } Convert(in := "DB20_DisplaySysdata".dbw42, out => #DWTemp2)
   END_RUNG
   // the same network as SCL:
   IF "On" THEN
       #DWTemp1 := INT_TO_DINT("DB04_Conveyor".dbw10);
       #DWTemp2 := INT_TO_DINT("DB20_DisplaySysdata".dbw42);
   END_IF;
END_REGION

REGION Network 10
   RUNG wire#powerrail
      Contact( "On" )
      { S7_Templates := "SrcType := DInt"; S7_GenerateENO := "TRUE" } Mul(in1 := #DWTemp1, in2 := #DWTemp2, out => #DWTemp1)
      { S7_Templates := "SrcType := DInt"; S7_GenerateENO := "TRUE" } Div(in1 := #DWTemp1, in2 := DINT#100, out => #DWTemp2)
   END_RUNG
   // the same network as SCL:
   // ENO of a box is taken as its EN; it also drops when the box reports an error
   IF "On" THEN
       #DWTemp1 := #DWTemp1 * #DWTemp2;
       #DWTemp2 := #DWTemp1 / DINT#100;
   END_IF;
END_REGION

REGION Network 11
   RUNG wire#powerrail
      { S7_GenerateENO := "TRUE" } Move(in := #DWTemp2, out1 => "DB04_Conveyor".dbw14)
   END_RUNG
   // the same network as SCL:
   "DB04_Conveyor".dbw14 := #DWTemp2;
END_REGION

REGION Network 12
   RUNG wire#powerrail
      Contact( "On" )
      wire#w1
      { S7_Templates := "[SrcType := Int, DestType := DInt]"; S7_GenerateENO := "TRUE" } Convert(in := "DB04_Conveyor".dbw12, out => #DWTemp1)
   END_RUNG
   RUNG wire#w1
      { S7_Templates := "[SrcType := Int, DestType := DInt]"; S7_GenerateENO := "TRUE" } Convert(in := "DB20_DisplaySysdata".dbw42, out => #DWTemp2)
   END_RUNG
   // the same network as SCL:
   IF "On" THEN
       #DWTemp1 := INT_TO_DINT("DB04_Conveyor".dbw12);
       #DWTemp2 := INT_TO_DINT("DB20_DisplaySysdata".dbw42);
   END_IF;
END_REGION

REGION Network 13
   RUNG wire#powerrail
      Contact( "On" )
      { S7_Templates := "SrcType := DInt"; S7_GenerateENO := "TRUE" } Mul(in1 := #DWTemp1, in2 := #DWTemp2, out => #DWTemp1)
      { S7_Templates := "SrcType := DInt"; S7_GenerateENO := "TRUE" } Div(in1 := #DWTemp1, in2 := DINT#100, out => #DWTemp2)
   END_RUNG
   // the same network as SCL:
   // ENO of a box is taken as its EN; it also drops when the box reports an error
   IF "On" THEN
       #DWTemp1 := #DWTemp1 * #DWTemp2;
       #DWTemp2 := #DWTemp1 / DINT#100;
   END_IF;
END_REGION

REGION Network 14
